// TIA Portal project "PLC_TEST_PROJECT_1" (V16)

(* hardware
DEVICE "S71500/ET200MP station_1"  S7-1500 station
   slot 0: "Rail_0"  Rack  6ES7 590-1***0-0AA0
   slot 1: "PLC_1"  CPU 1518F-4 PN/DP  6ES7 518-4FP00-0AB0  V2.8
      slot 3: "CPU display_1"  6ES7591-1BA00-0AA0
      slot 32768: "PROFINET interface_1"  X1
         slot 32769: "Port_1"  X1 P1
         slot 32770: "Port_2"  X1 P2
      slot 33024: "PROFINET interface_2"  X2
         slot 33025: "Port_1"  X2 P1
      slot 33280: "PROFINET interface GBIT_3"  X3
         slot 33281: "Port_1"  X3 P1
      slot 33536: "DP interface_1"  X4
      slot 34817: "Virtual CP interface port_1"  Virtual CP interface port  Virtual CP interface port
DEVICE "PCSTATION"  SIMATIC PC station
   slot 0: "PC station"  Rail  SIMATIC PC-Station  V1.0
      slot 125: "Stationmanager"  Station_Manager  V6.0.4
   slot 2: "HMI_RT_1"  WinCC RT Professional  6AV2 105-0xxxx-xxxx  16.0.0.0
*)

// ===== PLC "PLC_1"  CPU 1518F-4 PN/DP =====

VAR_GLOBAL   // PLC tag table "Default tag table"
   "Clock_Byte" AT %MB0 : Byte;
   "Clock_10Hz" AT %M0.0 : Bool;
   "Clock_5Hz" AT %M0.1 : Bool;
   "Clock_2.5Hz" AT %M0.2 : Bool;
   "Clock_2Hz" AT %M0.3 : Bool;
   "Clock_1.25Hz" AT %M0.4 : Bool;
   "Clock_1Hz" AT %M0.5 : Bool;
   "Clock_0.625Hz" AT %M0.6 : Bool;
   "Clock_0.5Hz" AT %M0.7 : Bool;
   "Tag_1" AT %MD104 : DWord;
   "Tag_2" AT %MD100 : DWord;
END_VAR

// folder: Common

TYPE "typeDiagnostics"
TITLE = typeDiagnostics
// Provides a structure for detailed diagnostics
   STRUCT
      status : Word;   // Status of the block or error identification when error occurred
      subfunctionStatus : DWord;   // Status or return value of called FBs, FCs and system blocks
      stateNumber : DInt;   // State in the state machine of the block where the error occurred
   END_STRUCT;
END_TYPE

// folder: LMQTT

TYPE "LMQTT_typeConnParam"
TITLE = LMQTT_typeConnParams
// Specifies connection parameters for the mqtt connection
   STRUCT
      hwId : Hw_Any;   // Hardware identifier of the interface. 0: interface is selected automatically
      connId : Conn_Ouc;   // Unique connection identifier
      brokerAddress : Struct   // Information on the MQTT broker
         qdnAddress : String;   // Fully qualified domain name of the broker. must end with a dot "."
         ipAddress : IP_V4;   // If no FQDN is used, enter ip-address of the broker instead
         port : UInt;   // Enter the port of the mqtt broker
      END_STRUCT;
      tls : Struct   // Parameters for TLS encryption
         enableTls : Bool;   // TRUE: Enables TLS, FALSE: disable TLS
         validateServerIdentity : Bool;   // TRUE: Validate server certificate, FALSE: No validation of server certificate
         brokerCert : UDInt;   // ID of the broker's certificate in TIA Portal
         clientCert : UDInt;   // ID of the client's certificate in TIA Portal
      END_STRUCT;
      keepAlive : UInt;   // Keepalive mechanism for MQTT in seconds. 0: disabled.
   END_STRUCT;
END_TYPE

// folder: (top level)

DATA_BLOCK "Main_Safety_RTG1_DB"   // DB1, F_DB
{ S7_Optimized_Access := 'TRUE' }
NAME : FUSI
VERSION : 0.1
// stored: InstanceOfName Main_Safety_RTG1
"Main_Safety_RTG1"
BEGIN
END_DATA_BLOCK

DATA_BLOCK "Timers"   // DB7
{ S7_Optimized_Access := 'TRUE' }
VERSION : 0.1
   VAR
      ElapsedTime : Time;
   END_VAR
BEGIN
END_DATA_BLOCK

DATA_BLOCK "DB_CMD"   // DB100
{ S7_Optimized_Access := 'FALSE' }
VERSION : 0.1
   VAR
      CMD_BOOL_1 : Bool;
      CMD_BOOL_2 : Bool;
      CMD_BOOL_3 : Bool;
      CMD_BOOL_4 : Bool;
      CMD_BOOL_5 : Bool;
      EnableCyclicPub : Bool;
      EnableTimeFrame : Bool;
      CMD_BOOL_8 : Bool;
      CMD_BOOL_9 : Bool;
      CMD_BOOL_10 : Bool;
      EnableCounter : Bool;
      EnableCounter4 : Bool;
      EnableCounter6 : Bool;
      EnableCounter10 : Bool;
   END_VAR
BEGIN
END_DATA_BLOCK

DATA_BLOCK "DB_STATUS"   // DB200
{ S7_Optimized_Access := 'FALSE' }
VERSION : 0.1
   VAR
      STAT_INT_1 : Int;
      STAT_INT_2 : Int;
      STAT_INT_3 : Int;
      STAT_INT_4 : Int;
      STAT_INT_5 : Int;
      STAT_INT_6 : Int;
      STAT_INT_7 : Int;
      STAT_INT_8 : Int;
      STAT_INT_9 : Int;
      STAT_INT_10 : Int;
      STAT_DINT_1 : DInt;
      STAT_DINT_2 : DInt;
      STAT_DINT_3 : DInt;
      STAT_DINT_4 : DInt;
      STAT_DINT_5 : DInt;
      STAT_DINT_6 : DInt;
      STAT_DINT_7 : DInt;
      STAT_DINT_8 : DInt;
      STAT_DINT_9 : DInt;
      STAT_DINT_10 : DInt;
      STAT_BOOL_1 : Bool;
      STAT_BOOL_2 : Bool;
      STAT_BOOL_3 : Bool;
      STAT_BOOL_4 : Bool;
      STAT_BOOL_5 : Bool;
      STAT_BOOL_6 : Bool;
      STAT_BOOL_7 : Bool;
      STAT_BOOL_8 : Bool;
      STAT_BOOL_9 : Bool;
      STAT_BOOL_10 : Bool;
      STAT_WCHAR_1 : Array[0..9] of Char;
   END_VAR
BEGIN
   STAT_WCHAR_1[0] := 'c';
   STAT_WCHAR_1[1] := 'b';
   STAT_WCHAR_1[2] := 'c';
END_DATA_BLOCK

DATA_BLOCK "DB_STATUS_CHECK"   // DB201
{ S7_Optimized_Access := 'FALSE' }
VERSION : 0.1
   VAR
      STAT_INT_1 : Int;
      STAT_INT_2 : Int;
      STAT_INT_3 : Int;
      STAT_INT_4 : Int;
      STAT_INT_5 : Int;
      STAT_INT_6 : Int;
      STAT_INT_7 : Int;
      STAT_INT_8 : Int;
      STAT_INT_9 : Int;
      STAT_INT_10 : Int;
      STAT_DINT_1 : DInt;
      STAT_DINT_2 : DInt;
      STAT_DINT_3 : DInt;
      STAT_DINT_4 : DInt;
      STAT_DINT_5 : DInt;
      STAT_DINT_6 : DInt;
      STAT_DINT_7 : DInt;
      STAT_DINT_8 : DInt;
      STAT_DINT_9 : DInt;
      STAT_DINT_10 : DInt;
      STAT_BOOL_1 : Bool;
      STAT_BOOL_2 : Bool;
      STAT_BOOL_3 : Bool;
      STAT_BOOL_4 : Bool;
      STAT_BOOL_5 : Bool;
      STAT_BOOL_6 : Bool;
      STAT_BOOL_7 : Bool;
      STAT_BOOL_8 : Bool;
      STAT_BOOL_9 : Bool;
      STAT_BOOL_10 : Bool;
      STAT_WCHAR_1 : Array[0..9] of Char;
   END_VAR
BEGIN
   STAT_WCHAR_1[0] := 'c';
   STAT_WCHAR_1[1] := 'b';
   STAT_WCHAR_1[2] := 'c';
END_DATA_BLOCK

DATA_BLOCK "DB_STATUS_ADDR_BYTE"   // DB202
{ S7_Optimized_Access := 'FALSE' }
VERSION : 0.1
   VAR
      STAT_INT_1 : Int := 0;
      STAT_INT_2 : Int := 2;
      STAT_INT_3 : Int := 4;
      STAT_INT_4 : Int := 6;
      STAT_INT_5 : Int := 8;
      STAT_INT_6 : Int := 10;
      STAT_INT_7 : Int := 12;
      STAT_INT_8 : Int := 14;
      STAT_INT_9 : Int := 16;
      STAT_INT_10 : Int := 18;
      STAT_DINT_1 : Int := 20;
      STAT_DINT_2 : Int := 24;
      STAT_DINT_3 : Int := 28;
      STAT_DINT_4 : Int := 32;
      STAT_DINT_5 : Int := 36;
      STAT_DINT_6 : Int := 40;
      STAT_DINT_7 : Int := 44;
      STAT_DINT_8 : Int := 48;
      STAT_DINT_9 : Int := 52;
      STAT_DINT_10 : Int := 56;
      STAT_BOOL_1 : Int := 60;
      STAT_BOOL_2 : Int := 60;
      STAT_BOOL_3 : Int := 60;
      STAT_BOOL_4 : Int := 60;
      STAT_BOOL_5 : Int := 60;
      STAT_BOOL_6 : Int := 60;
      STAT_BOOL_7 : Int := 60;
      STAT_BOOL_8 : Int := 60;
      STAT_BOOL_9 : Int := 61;
      STAT_BOOL_10 : Int := 61;
      STAT_WCHAR_1 : Int := 62;
   END_VAR
BEGIN
END_DATA_BLOCK

DATA_BLOCK "DB_STATUS_ADDR_BIT"   // DB203
{ S7_Optimized_Access := 'FALSE' }
VERSION : 0.1
   VAR
      STAT_INT_1 : Byte := 0;
      STAT_INT_2 : Byte := 0;
      STAT_INT_3 : Byte := 0;
      STAT_INT_4 : Byte := 0;
      STAT_INT_5 : Byte := 0;
      STAT_INT_6 : Byte := 0;
      STAT_INT_7 : Byte := 0;
      STAT_INT_8 : Byte := 0;
      STAT_INT_9 : Byte := 0;
      STAT_INT_10 : Byte := 0;
      STAT_DINT_1 : Byte := 0;
      STAT_DINT_2 : Byte := 0;
      STAT_DINT_3 : Byte := 0;
      STAT_DINT_4 : Byte := 0;
      STAT_DINT_5 : Byte := 0;
      STAT_DINT_6 : Byte := 0;
      STAT_DINT_7 : Byte := 0;
      STAT_DINT_8 : Byte := 0;
      STAT_DINT_9 : Byte := 0;
      STAT_DINT_10 : Byte := 0;
      STAT_BOOL_1 : Byte := 0;
      STAT_BOOL_2 : Byte := 1;
      STAT_BOOL_3 : Byte := 2;
      STAT_BOOL_4 : Byte := 3;
      STAT_BOOL_5 : Byte := 4;
      STAT_BOOL_6 : Byte := 5;
      STAT_BOOL_7 : Byte := 6;
      STAT_BOOL_8 : Byte := 7;
      STAT_BOOL_9 : Byte := 0;
      STAT_BOOL_10 : Byte := 0;
      STAT_WCHAR_1 : Byte := 10;
   END_VAR
BEGIN
END_DATA_BLOCK

// folder: DataChange

DATA_BLOCK "DB_DataChange"   // DB5
{ S7_Optimized_Access := 'FALSE' }
VERSION : 0.1
   VAR
      StartMQTT : Bool;
      DataChanged : Bool;
      DataTypeCode : Array[0..0] of Byte;
   END_VAR
BEGIN
END_DATA_BLOCK

// folder: LMQTT

DATA_BLOCK "LMQTT_Client_DB"   // DB2
{ S7_Optimized_Access := 'TRUE' }
AUTHOR : SUP
FAMILY : LMQTT
VERSION : 3.0
// stored: InstanceOfName LMQTT_Client
"LMQTT_Client"
BEGIN
END_DATA_BLOCK

DATA_BLOCK "MqttDb"   // DB3
TITLE = Configuration Data block example for LMQTT_Client
{ S7_Optimized_Access := 'TRUE' }
AUTHOR : Siemens
FAMILY : LMQTT
VERSION : 1.0
// This block is an example how to control the LMQTT_Client function block
   VAR
      control : Struct   // Input of the FB
         connect : Bool;   // Set TRUE, to establish a connection - set to FALSE to disconnect
         publish : Bool;   // Rising Edge: Sends a message
         subscribe : Bool;   // Rising Edge: Subscribes to a topic
         unsubscribe : Bool;   // Rising Edge: Unsubscribes to a topic
      END_STRUCT;
      output : Struct   // Output Information of the FB
         valid : Bool;   // TRUE: Valid set of output values available at the FB
         done : Bool;   // TRUE: If last Request was successfull
         busy : Bool;   // TRUE: FB is not finished and new output values can be expected
         error : Bool;   // TRUE: An error occurred during the execution of the FB
         status : Word;   // 16#0000 - 16#7FFF: Status of the FB, 16#8000 - 16#FFFF: Error identification
         diagnostics : "typeDiagnostics";   // Diagnostics information of FB (optional)
      END_STRUCT;
      connparams : "LMQTT_typeConnParam";   // Connection Parameters
      clientid : WString[20] := WSTRING#'SiemensClient';   // ClientId with one or more characters
      username : WString[20];   // Username used for connect
      password : WString[20];   // Password used for connect
      willtopic : WString[20] := WSTRING#'willTopic';   // Topic where the last will message is sent
      willMessage : Array[0..99] of Byte;   // Last will message Data - valid bytes in this array must be written in input 'willMsgLen'
      willmesscnt : UInt := 10;   // Valid number of elements in Will Message Data Array. Max 65535 Byte allowed by MQTT Spec.
      qos : USInt := 0;   // Sets QoS 0,1 or 2 for the Publish and Will Message - Subscribe only allows QoS 0 and 1
      topic : WString[100] := WSTRING#'TIA-test-project';   // Mqtt Topic to Publish / Subscribe / Unsubscribe
      message : Array[0..99] of Byte;   // Message Data to Publish - valid bytes in this array must be written in input 'publishMsgLen'
      pubMessageCnt : UDInt := 11;   // Valid number of elements in publish message data Array
      retain : Bool;   // TRUE: Published Message will be set to retain on MQTT broker
      receivedTopic : WString[200] := WSTRING#'TIA-test-project';   // Mqtt Topic of received message
      receivedmessage : Array[0..99] of Byte;   // Mqtt message data that was received - valid bytes in this array indicated by 'receivedMsgDataLen' output
      receivedMsgLen : UDInt;   // Amount of Bytes received in receivedMessage INOUT area
      receivedMsgStatus : USInt;   // 0: No new Message, 1: New valid Message received and available at InOut area, 2: New message, but data is invalid (wrong message len or message could not be copied to InOut received topic or received message)
   END_VAR
BEGIN
   willMessage[0] := 16#6F;
   willMessage[1] := 16#66;
   willMessage[2] := 16#66;
   willMessage[3] := 16#6C;
   willMessage[4] := 16#69;
   willMessage[5] := 16#6E;
   willMessage[6] := 16#65;
   message[1] := 16#65;
   message[2] := 16#6c;
   message[3] := 16#6c;
   message[4] := 16#6f;
   message[5] := 16#20;
   message[6] := 16#77;
   message[7] := 16#6f;
   message[8] := 16#72;
   message[9] := 16#6c;
   message[10] := 16#64;
   message[0] := 16#68;
   connparams.connId := 16#10;
   connparams.brokerAddress.ipAddress.ADDR[1] := 192;
   connparams.brokerAddress.ipAddress.ADDR[2] := 168;
   connparams.brokerAddress.ipAddress.ADDR[3] := 0;
   connparams.brokerAddress.ipAddress.ADDR[4] := 250;
   connparams.brokerAddress.port := 1883;
   connparams.hwId := 64;
   connparams.keepAlive := 100;
END_DATA_BLOCK

// folder: MQTT_pub

DATA_BLOCK "DB_MQTT_PUB"   // DB4
{ S7_Optimized_Access := 'FALSE' }
VERSION : 0.1
   VAR
      DataTypeCodeTemp : Array[0..0] of Byte;
   END_VAR
BEGIN
END_DATA_BLOCK

// folder: Serialize

DATA_BLOCK "DB_Serialize"   // DB1001
{ S7_Optimized_Access := 'TRUE' }
VERSION : 0.1
   VAR
      SERIAL_BYTEARRAY : Array[0..99] of Byte;
      SER_ERROR_CODE : Int;
      SER_START_INDEX : Int;
   END_VAR
BEGIN
END_DATA_BLOCK

// folder: System blocks/Program resources

DATA_BLOCK "TrigDelay"   // DB6
{ S7_Optimized_Access := 'TRUE' }
AUTHOR : Simatic
FAMILY : IEC
NAME : IEC_TMR
VERSION : 1.0
// stored: InstanceOfName IEC_TIMER
"IEC_TIMER"
BEGIN
END_DATA_BLOCK

DATA_BLOCK "IncrementTimer"   // DB8
{ S7_Optimized_Access := 'TRUE' }
AUTHOR : Simatic
FAMILY : IEC
NAME : IEC_TMR
VERSION : 1.0
// stored: InstanceOfName IEC_TIMER
"IEC_TIMER"
BEGIN
END_DATA_BLOCK

// folder: (top level)

FUNCTION_BLOCK "Main_Safety_RTG1"   // FB1, F_FBD
{ S7_Optimized_Access := 'TRUE' }
BEGIN
END_FUNCTION_BLOCK

FUNCTION "DataChange" : Void   // FC3, SCL
{ S7_Optimized_Access := 'TRUE' }
VERSION : 0.1
   VAR_OUTPUT
      DataChanged : Bool;
   END_VAR
   VAR_TEMP
      i : Int;
      TagChanged : Int;
      DataTypeBytelen : Int;
   END_VAR
BEGIN
   (*

   *)

   IF "DB_STATUS".STAT_INT_1 <> "DB_STATUS_CHECK".STAT_INT_1 THEN
       "DB_STATUS_CHECK".STAT_INT_1 := "DB_STATUS".STAT_INT_1;

       //Serialize address byte  - first 4 bytes in MQTT message array [0,1,2,3]
       "Serialize_to_ByteArray"(StartIndexOutputArray := "DB_Serialize".SER_START_INDEX,
                                Input_tag_any_type := "DB_STATUS_ADDR_BYTE".STAT_INT_1,
                                OutputArray => "MqttDb".message,
                                RetVal_error => "DB_Serialize".SER_ERROR_CODE);
       "DB_Serialize".SER_START_INDEX :=  "DB_Serialize".SER_START_INDEX + 4;

       //Serialize address bit (or array length) -  next 1 byte in MQTT message array [4]
       "Serialize_to_ByteArray"(StartIndexOutputArray := "DB_Serialize".SER_START_INDEX,
                                Input_tag_any_type := "DB_STATUS_ADDR_BIT".STAT_INT_1,
                                OutputArray => "MqttDb".message,
                                RetVal_error => "DB_Serialize".SER_ERROR_CODE);
       "DB_Serialize".SER_START_INDEX := "DB_Serialize".SER_START_INDEX + 1;

       //Serialize data type -  next 1 byte in MQTT message array [5]
       "GetDataTypeCode"(DataTypeByteLen=>#DataTypeBytelen,
                         DataTypeCode => "DB_DataChange".DataTypeCode,
                         InOutVariant := "DB_STATUS".STAT_INT_1);
       "MqttDb".message["DB_Serialize".SER_START_INDEX] := "DB_DataChange".DataTypeCode[0];
       "DB_Serialize".SER_START_INDEX := "DB_Serialize".SER_START_INDEX + 1;

       //Serialize tag value -  next 1 byte in MQTT message array [6]
       "Serialize_to_ByteArray"(StartIndexOutputArray := "DB_Serialize".SER_START_INDEX,
                                Input_tag_any_type := "DB_STATUS".STAT_INT_1,
                                OutputArray => "MqttDb".message,
                                RetVal_error => "DB_Serialize".SER_ERROR_CODE);
       //Set index for next tag in MQTT message array
       "DB_Serialize".SER_START_INDEX := "DB_Serialize".SER_START_INDEX + #DataTypeBytelen;
       #TagChanged := #TagChanged + 1;
   END_IF;

   IF "DB_STATUS".STAT_INT_2 <> "DB_STATUS_CHECK".STAT_INT_2 THEN
       "DB_STATUS_CHECK".STAT_INT_2 := "DB_STATUS".STAT_INT_2;

       //Serialize address byte  - first 4 bytes in MQTT message array [0,1,2,3]
       "Serialize_to_ByteArray"(StartIndexOutputArray := "DB_Serialize".SER_START_INDEX,
                                Input_tag_any_type := "DB_STATUS_ADDR_BYTE".STAT_INT_2,
                                OutputArray => "MqttDb".message,
                                RetVal_error => "DB_Serialize".SER_ERROR_CODE);
       "DB_Serialize".SER_START_INDEX := "DB_Serialize".SER_START_INDEX + 4;

       //Serialize address bit (or array length) -  next 1 byte in MQTT message array [4]
       "Serialize_to_ByteArray"(StartIndexOutputArray := "DB_Serialize".SER_START_INDEX,
                                Input_tag_any_type := "DB_STATUS_ADDR_BIT".STAT_INT_2,
                                OutputArray => "MqttDb".message,
                                RetVal_error => "DB_Serialize".SER_ERROR_CODE);
       "DB_Serialize".SER_START_INDEX := "DB_Serialize".SER_START_INDEX + 1;

       //Serialize data type -  next 1 byte in MQTT message array [5]
       "GetDataTypeCode"(DataTypeByteLen => #DataTypeBytelen,
                         DataTypeCode => "DB_DataChange".DataTypeCode,
                         InOutVariant := "DB_STATUS".STAT_INT_2);
       "MqttDb".message["DB_Serialize".SER_START_INDEX] := "DB_DataChange".DataTypeCode[0];
       "DB_Serialize".SER_START_INDEX := "DB_Serialize".SER_START_INDEX + 1;

       //Serialize tag value -  next 1 byte in MQTT message array [6]
       "Serialize_to_ByteArray"(StartIndexOutputArray := "DB_Serialize".SER_START_INDEX,
                                Input_tag_any_type := "DB_STATUS".STAT_INT_2,
                                OutputArray => "MqttDb".message,
                                RetVal_error => "DB_Serialize".SER_ERROR_CODE);
       //Set index for next tag in MQTT message array
       "DB_Serialize".SER_START_INDEX := "DB_Serialize".SER_START_INDEX + #DataTypeBytelen;
       #TagChanged := #TagChanged + 1;
   END_IF;

   IF "DB_STATUS".STAT_INT_3 <> "DB_STATUS_CHECK".STAT_INT_3 THEN
       "DB_STATUS_CHECK".STAT_INT_3 := "DB_STATUS".STAT_INT_3;

       //Serialize address byte  - first 4 bytes in MQTT message array [0,1,2,3]
       "Serialize_to_ByteArray"(StartIndexOutputArray := "DB_Serialize".SER_START_INDEX,
                                Input_tag_any_type := "DB_STATUS_ADDR_BYTE".STAT_INT_3,
                                OutputArray => "MqttDb".message,
                                RetVal_error => "DB_Serialize".SER_ERROR_CODE);
       "DB_Serialize".SER_START_INDEX := "DB_Serialize".SER_START_INDEX + 4;

       //Serialize address bit (or array length) -  next 1 byte in MQTT message array [4]
       "Serialize_to_ByteArray"(StartIndexOutputArray := "DB_Serialize".SER_START_INDEX,
                                Input_tag_any_type := "DB_STATUS_ADDR_BIT".STAT_INT_3,
                                OutputArray => "MqttDb".message,
                                RetVal_error => "DB_Serialize".SER_ERROR_CODE);
       "DB_Serialize".SER_START_INDEX := "DB_Serialize".SER_START_INDEX + 1;

       //Serialize data type -  next 1 byte in MQTT message array [5]
       "GetDataTypeCode"(DataTypeByteLen => #DataTypeBytelen,
                         DataTypeCode => "DB_DataChange".DataTypeCode,
                         InOutVariant := "DB_STATUS".STAT_INT_3);
       "MqttDb".message["DB_Serialize".SER_START_INDEX] := "DB_DataChange".DataTypeCode[0];
       "DB_Serialize".SER_START_INDEX := "DB_Serialize".SER_START_INDEX + 1;

       //Serialize tag value -  next 1 byte in MQTT message array [6]
       "Serialize_to_ByteArray"(StartIndexOutputArray := "DB_Serialize".SER_START_INDEX,
                                Input_tag_any_type := "DB_STATUS".STAT_INT_3,
                                OutputArray => "MqttDb".message,
                                RetVal_error => "DB_Serialize".SER_ERROR_CODE);
       //Set index for next tag in MQTT message array
       "DB_Serialize".SER_START_INDEX := "DB_Serialize".SER_START_INDEX + #DataTypeBytelen;
       #TagChanged := #TagChanged + 1;
   END_IF;

   IF "DB_STATUS".STAT_INT_4 <> "DB_STATUS_CHECK".STAT_INT_4 THEN
       "DB_STATUS_CHECK".STAT_INT_4 := "DB_STATUS".STAT_INT_4;

       //Serialize address byte  - first 4 bytes in MQTT message array [0,1,2,3]
       "Serialize_to_ByteArray"(StartIndexOutputArray := "DB_Serialize".SER_START_INDEX,
                                Input_tag_any_type := "DB_STATUS_ADDR_BYTE".STAT_INT_4,
                                OutputArray => "MqttDb".message,
                                RetVal_error => "DB_Serialize".SER_ERROR_CODE);
       "DB_Serialize".SER_START_INDEX := "DB_Serialize".SER_START_INDEX + 4;

       //Serialize address bit (or array length) -  next 1 byte in MQTT message array [4]
       "Serialize_to_ByteArray"(StartIndexOutputArray := "DB_Serialize".SER_START_INDEX,
                                Input_tag_any_type := "DB_STATUS_ADDR_BIT".STAT_INT_4,
                                OutputArray => "MqttDb".message,
                                RetVal_error => "DB_Serialize".SER_ERROR_CODE);
       "DB_Serialize".SER_START_INDEX := "DB_Serialize".SER_START_INDEX + 1;

       //Serialize data type -  next 1 byte in MQTT message array [5]
       "GetDataTypeCode"(DataTypeByteLen => #DataTypeBytelen,
                         DataTypeCode => "DB_DataChange".DataTypeCode,
                         InOutVariant := "DB_STATUS".STAT_INT_4);
       "MqttDb".message["DB_Serialize".SER_START_INDEX] := "DB_DataChange".DataTypeCode[0];
       "DB_Serialize".SER_START_INDEX := "DB_Serialize".SER_START_INDEX + 1;

       //Serialize tag value -  next 1 byte in MQTT message array [6]
       "Serialize_to_ByteArray"(StartIndexOutputArray := "DB_Serialize".SER_START_INDEX,
                                Input_tag_any_type := "DB_STATUS".STAT_INT_4,
                                OutputArray => "MqttDb".message,
                                RetVal_error => "DB_Serialize".SER_ERROR_CODE);
       //Set index for next tag in MQTT message array
       "DB_Serialize".SER_START_INDEX := "DB_Serialize".SER_START_INDEX + #DataTypeBytelen;
       #TagChanged := #TagChanged + 1;
   END_IF;

   IF "DB_STATUS".STAT_INT_5 <> "DB_STATUS_CHECK".STAT_INT_5 THEN
       "DB_STATUS_CHECK".STAT_INT_5 := "DB_STATUS".STAT_INT_5;

       //Serialize address byte  - first 4 bytes in MQTT message array [0,1,2,3]
       "Serialize_to_ByteArray"(StartIndexOutputArray := "DB_Serialize".SER_START_INDEX,
                                Input_tag_any_type := "DB_STATUS_ADDR_BYTE".STAT_INT_5,
                                OutputArray => "MqttDb".message,
                                RetVal_error => "DB_Serialize".SER_ERROR_CODE);
       "DB_Serialize".SER_START_INDEX := "DB_Serialize".SER_START_INDEX + 4;

       //Serialize address bit (or array length) -  next 1 byte in MQTT message array [4]
       "Serialize_to_ByteArray"(StartIndexOutputArray := "DB_Serialize".SER_START_INDEX,
                                Input_tag_any_type := "DB_STATUS_ADDR_BIT".STAT_INT_5,
                                OutputArray => "MqttDb".message,
                                RetVal_error => "DB_Serialize".SER_ERROR_CODE);
       "DB_Serialize".SER_START_INDEX := "DB_Serialize".SER_START_INDEX + 1;

       //Serialize data type -  next 1 byte in MQTT message array [5]
       "GetDataTypeCode"(DataTypeByteLen => #DataTypeBytelen,
                         DataTypeCode => "DB_DataChange".DataTypeCode,
                         InOutVariant := "DB_STATUS".STAT_INT_5);
       "MqttDb".message["DB_Serialize".SER_START_INDEX] := "DB_DataChange".DataTypeCode[0];
       "DB_Serialize".SER_START_INDEX := "DB_Serialize".SER_START_INDEX + 1;

       //Serialize tag value -  next 1 byte in MQTT message array [6]
       "Serialize_to_ByteArray"(StartIndexOutputArray := "DB_Serialize".SER_START_INDEX,
                                Input_tag_any_type := "DB_STATUS".STAT_INT_5,
                                OutputArray => "MqttDb".message,
                                RetVal_error => "DB_Serialize".SER_ERROR_CODE);
       //Set index for next tag in MQTT message array
       "DB_Serialize".SER_START_INDEX := "DB_Serialize".SER_START_INDEX + #DataTypeBytelen;
       #TagChanged := #TagChanged + 1;
   END_IF;

   IF "DB_STATUS".STAT_DINT_1 <> "DB_STATUS_CHECK".STAT_DINT_1 THEN
       "DB_STATUS_CHECK".STAT_DINT_1 := "DB_STATUS".STAT_DINT_1;

       //Serialize address byte  - first 4 bytes in MQTT message array [0,1,2,3]
       "Serialize_to_ByteArray"(StartIndexOutputArray := "DB_Serialize".SER_START_INDEX,
                                Input_tag_any_type := "DB_STATUS_ADDR_BYTE".STAT_DINT_1,
                                OutputArray => "MqttDb".message,
                                RetVal_error => "DB_Serialize".SER_ERROR_CODE);
       "DB_Serialize".SER_START_INDEX := "DB_Serialize".SER_START_INDEX + 4;

       //Serialize address bit (or array length) -  next 1 byte in MQTT message array [4]
       "Serialize_to_ByteArray"(StartIndexOutputArray := "DB_Serialize".SER_START_INDEX,
                                Input_tag_any_type := "DB_STATUS_ADDR_BIT".STAT_DINT_1,
                                OutputArray => "MqttDb".message,
                                RetVal_error => "DB_Serialize".SER_ERROR_CODE);
       "DB_Serialize".SER_START_INDEX := "DB_Serialize".SER_START_INDEX + 1;

       //Serialize data type -  next 1 byte in MQTT message array [5]
       "GetDataTypeCode"(DataTypeByteLen => #DataTypeBytelen,
                         DataTypeCode => "DB_DataChange".DataTypeCode,
                         InOutVariant := "DB_STATUS".STAT_DINT_1);
       "MqttDb".message["DB_Serialize".SER_START_INDEX] := "DB_DataChange".DataTypeCode[0];
       "DB_Serialize".SER_START_INDEX := "DB_Serialize".SER_START_INDEX + 1;

       //Serialize tag value -  next 1 byte in MQTT message array [6]
       "Serialize_to_ByteArray"(StartIndexOutputArray := "DB_Serialize".SER_START_INDEX,
                                Input_tag_any_type := "DB_STATUS".STAT_DINT_1,
                                OutputArray => "MqttDb".message,
                                RetVal_error => "DB_Serialize".SER_ERROR_CODE);
       //Set index for next tag in MQTT message array
       "DB_Serialize".SER_START_INDEX := "DB_Serialize".SER_START_INDEX + #DataTypeBytelen;
       #TagChanged := #TagChanged + 1;
   END_IF;

   IF "DB_STATUS".STAT_DINT_2 <> "DB_STATUS_CHECK".STAT_DINT_2 THEN
       "DB_STATUS_CHECK".STAT_DINT_2 := "DB_STATUS".STAT_DINT_2;

       //Serialize address byte  - first 4 bytes in MQTT message array [0,1,2,3]
       "Serialize_to_ByteArray"(StartIndexOutputArray := "DB_Serialize".SER_START_INDEX,
                                Input_tag_any_type := "DB_STATUS_ADDR_BYTE".STAT_DINT_2,
                                OutputArray => "MqttDb".message,
                                RetVal_error => "DB_Serialize".SER_ERROR_CODE);
       "DB_Serialize".SER_START_INDEX := "DB_Serialize".SER_START_INDEX + 4;

       //Serialize address bit (or array length) -  next 1 byte in MQTT message array [4]
       "Serialize_to_ByteArray"(StartIndexOutputArray := "DB_Serialize".SER_START_INDEX,
                                Input_tag_any_type := "DB_STATUS_ADDR_BIT".STAT_DINT_2,
                                OutputArray => "MqttDb".message,
                                RetVal_error => "DB_Serialize".SER_ERROR_CODE);
       "DB_Serialize".SER_START_INDEX := "DB_Serialize".SER_START_INDEX + 1;

       //Serialize data type -  next 1 byte in MQTT message array [5]
       "GetDataTypeCode"(DataTypeByteLen => #DataTypeBytelen,
                         DataTypeCode => "DB_DataChange".DataTypeCode,
                         InOutVariant := "DB_STATUS".STAT_DINT_2);
       "MqttDb".message["DB_Serialize".SER_START_INDEX] := "DB_DataChange".DataTypeCode[0];
       "DB_Serialize".SER_START_INDEX := "DB_Serialize".SER_START_INDEX + 1;

       //Serialize tag value -  next 1 byte in MQTT message array [6]
       "Serialize_to_ByteArray"(StartIndexOutputArray := "DB_Serialize".SER_START_INDEX,
                                Input_tag_any_type := "DB_STATUS".STAT_DINT_2,
                                OutputArray => "MqttDb".message,
                                RetVal_error => "DB_Serialize".SER_ERROR_CODE);
       //Set index for next tag in MQTT message array
       "DB_Serialize".SER_START_INDEX := "DB_Serialize".SER_START_INDEX + #DataTypeBytelen;
       #TagChanged := #TagChanged + 1;
   END_IF;

   IF "DB_STATUS".STAT_DINT_3 <> "DB_STATUS_CHECK".STAT_DINT_3 THEN
       "DB_STATUS_CHECK".STAT_DINT_3 := "DB_STATUS".STAT_DINT_3;

       //Serialize address byte  - first 4 bytes in MQTT message array [0,1,2,3]
       "Serialize_to_ByteArray"(StartIndexOutputArray := "DB_Serialize".SER_START_INDEX,
                                Input_tag_any_type := "DB_STATUS_ADDR_BYTE".STAT_DINT_3,
                                OutputArray => "MqttDb".message,
                                RetVal_error => "DB_Serialize".SER_ERROR_CODE);
       "DB_Serialize".SER_START_INDEX := "DB_Serialize".SER_START_INDEX + 4;

       //Serialize address bit (or array length) -  next 1 byte in MQTT message array [4]
       "Serialize_to_ByteArray"(StartIndexOutputArray := "DB_Serialize".SER_START_INDEX,
                                Input_tag_any_type := "DB_STATUS_ADDR_BIT".STAT_DINT_3,
                                OutputArray => "MqttDb".message,
                                RetVal_error => "DB_Serialize".SER_ERROR_CODE);
       "DB_Serialize".SER_START_INDEX := "DB_Serialize".SER_START_INDEX + 1;

       //Serialize data type -  next 1 byte in MQTT message array [5]
       "GetDataTypeCode"(DataTypeByteLen => #DataTypeBytelen,
                         DataTypeCode => "DB_DataChange".DataTypeCode,
                         InOutVariant := "DB_STATUS".STAT_DINT_3);
       "MqttDb".message["DB_Serialize".SER_START_INDEX] := "DB_DataChange".DataTypeCode[0];
       "DB_Serialize".SER_START_INDEX := "DB_Serialize".SER_START_INDEX + 1;

       //Serialize tag value -  next 1 byte in MQTT message array [6]
       "Serialize_to_ByteArray"(StartIndexOutputArray := "DB_Serialize".SER_START_INDEX,
                                Input_tag_any_type := "DB_STATUS".STAT_DINT_3,
                                OutputArray => "MqttDb".message,
                                RetVal_error => "DB_Serialize".SER_ERROR_CODE);
       //Set index for next tag in MQTT message array
       "DB_Serialize".SER_START_INDEX := "DB_Serialize".SER_START_INDEX + #DataTypeBytelen;
       #TagChanged := #TagChanged + 1;
   END_IF;

   IF "DB_STATUS".STAT_DINT_4 <> "DB_STATUS_CHECK".STAT_DINT_4 THEN
       "DB_STATUS_CHECK".STAT_DINT_4 := "DB_STATUS".STAT_DINT_4;

       //Serialize address byte  - first 4 bytes in MQTT message array [0,1,2,3]
       "Serialize_to_ByteArray"(StartIndexOutputArray := "DB_Serialize".SER_START_INDEX,
                                Input_tag_any_type := "DB_STATUS_ADDR_BYTE".STAT_DINT_4,
                                OutputArray => "MqttDb".message,
                                RetVal_error => "DB_Serialize".SER_ERROR_CODE);
       "DB_Serialize".SER_START_INDEX := "DB_Serialize".SER_START_INDEX + 4;

       //Serialize address bit (or array length) -  next 1 byte in MQTT message array [4]
       "Serialize_to_ByteArray"(StartIndexOutputArray := "DB_Serialize".SER_START_INDEX,
                                Input_tag_any_type := "DB_STATUS_ADDR_BIT".STAT_DINT_4,
                                OutputArray => "MqttDb".message,
                                RetVal_error => "DB_Serialize".SER_ERROR_CODE);
       "DB_Serialize".SER_START_INDEX := "DB_Serialize".SER_START_INDEX + 1;

       //Serialize data type -  next 1 byte in MQTT message array [5]
       "GetDataTypeCode"(DataTypeByteLen => #DataTypeBytelen,
                         DataTypeCode => "DB_DataChange".DataTypeCode,
                         InOutVariant := "DB_STATUS".STAT_DINT_4);
       "MqttDb".message["DB_Serialize".SER_START_INDEX] := "DB_DataChange".DataTypeCode[0];
       "DB_Serialize".SER_START_INDEX := "DB_Serialize".SER_START_INDEX + 1;

       //Serialize tag value -  next 1 byte in MQTT message array [6]
       "Serialize_to_ByteArray"(StartIndexOutputArray := "DB_Serialize".SER_START_INDEX,
                                Input_tag_any_type := "DB_STATUS".STAT_DINT_4,
                                OutputArray => "MqttDb".message,
                                RetVal_error => "DB_Serialize".SER_ERROR_CODE);
       //Set index for next tag in MQTT message array
       "DB_Serialize".SER_START_INDEX := "DB_Serialize".SER_START_INDEX + #DataTypeBytelen;
       #TagChanged := #TagChanged + 1;
   END_IF;

   IF "DB_STATUS".STAT_DINT_5 <> "DB_STATUS_CHECK".STAT_DINT_5 THEN
       "DB_STATUS_CHECK".STAT_DINT_5 := "DB_STATUS".STAT_DINT_5;

       //Serialize address byte  - first 4 bytes in MQTT message array [0,1,2,3]
       "Serialize_to_ByteArray"(StartIndexOutputArray := "DB_Serialize".SER_START_INDEX,
                                Input_tag_any_type := "DB_STATUS_ADDR_BYTE".STAT_DINT_5,
                                OutputArray => "MqttDb".message,
                                RetVal_error => "DB_Serialize".SER_ERROR_CODE);
       "DB_Serialize".SER_START_INDEX := "DB_Serialize".SER_START_INDEX + 4;

       //Serialize address bit (or array length) -  next 1 byte in MQTT message array [4]
       "Serialize_to_ByteArray"(StartIndexOutputArray := "DB_Serialize".SER_START_INDEX,
                                Input_tag_any_type := "DB_STATUS_ADDR_BIT".STAT_DINT_5,
                                OutputArray => "MqttDb".message,
                                RetVal_error => "DB_Serialize".SER_ERROR_CODE);
       "DB_Serialize".SER_START_INDEX := "DB_Serialize".SER_START_INDEX + 1;

       //Serialize data type -  next 1 byte in MQTT message array [5]
       "GetDataTypeCode"(DataTypeByteLen => #DataTypeBytelen,
                         DataTypeCode => "DB_DataChange".DataTypeCode,
                         InOutVariant := "DB_STATUS".STAT_DINT_5);
       "MqttDb".message["DB_Serialize".SER_START_INDEX] := "DB_DataChange".DataTypeCode[0];
       "DB_Serialize".SER_START_INDEX := "DB_Serialize".SER_START_INDEX + 1;

       //Serialize tag value -  next 1 byte in MQTT message array [6]
       "Serialize_to_ByteArray"(StartIndexOutputArray := "DB_Serialize".SER_START_INDEX,
                                Input_tag_any_type := "DB_STATUS".STAT_DINT_5,
                                OutputArray => "MqttDb".message,
                                RetVal_error => "DB_Serialize".SER_ERROR_CODE);
       //Set index for next tag in MQTT message array
       "DB_Serialize".SER_START_INDEX := "DB_Serialize".SER_START_INDEX + #DataTypeBytelen;
       #TagChanged := #TagChanged + 1;
   END_IF;

   IF "DB_STATUS".STAT_DINT_6 <> "DB_STATUS_CHECK".STAT_DINT_6 THEN
       "DB_STATUS_CHECK".STAT_DINT_6 := "DB_STATUS".STAT_DINT_6;

       //Serialize address byte  - first 4 bytes in MQTT message array [0,1,2,3]
       "Serialize_to_ByteArray"(StartIndexOutputArray := "DB_Serialize".SER_START_INDEX,
                                Input_tag_any_type := "DB_STATUS_ADDR_BYTE".STAT_DINT_6,
                                OutputArray => "MqttDb".message,
                                RetVal_error => "DB_Serialize".SER_ERROR_CODE);
       "DB_Serialize".SER_START_INDEX := "DB_Serialize".SER_START_INDEX + 4;

       //Serialize address bit (or array length) -  next 1 byte in MQTT message array [4]
       "Serialize_to_ByteArray"(StartIndexOutputArray := "DB_Serialize".SER_START_INDEX,
                                Input_tag_any_type := "DB_STATUS_ADDR_BIT".STAT_DINT_6,
                                OutputArray => "MqttDb".message,
                                RetVal_error => "DB_Serialize".SER_ERROR_CODE);
       "DB_Serialize".SER_START_INDEX := "DB_Serialize".SER_START_INDEX + 1;

       //Serialize data type -  next 1 byte in MQTT message array [5]
       "GetDataTypeCode"(DataTypeByteLen => #DataTypeBytelen,
                         DataTypeCode => "DB_DataChange".DataTypeCode,
                         InOutVariant := "DB_STATUS".STAT_DINT_6);
       "MqttDb".message["DB_Serialize".SER_START_INDEX] := "DB_DataChange".DataTypeCode[0];
       "DB_Serialize".SER_START_INDEX := "DB_Serialize".SER_START_INDEX + 1;

       //Serialize tag value -  next 1 byte in MQTT message array [6]
       "Serialize_to_ByteArray"(StartIndexOutputArray := "DB_Serialize".SER_START_INDEX,
                                Input_tag_any_type := "DB_STATUS".STAT_DINT_6,
                                OutputArray => "MqttDb".message,
                                RetVal_error => "DB_Serialize".SER_ERROR_CODE);
       //Set index for next tag in MQTT message array
       "DB_Serialize".SER_START_INDEX := "DB_Serialize".SER_START_INDEX + #DataTypeBytelen;
       #TagChanged := #TagChanged + 1;
   END_IF;

   //If any of the tags are changed, set output trigger.
   IF #TagChanged > 0 THEN
       "MqttDb".pubMessageCnt := "DB_Serialize".SER_START_INDEX; //Message array size
       "MqttDb".topic := WSTRING#'TIA-test-project/DB200';
       #DataChanged := TRUE;
   END_IF;
END_FUNCTION

ORGANIZATION_BLOCK "Main"   // OB1, LAD, ProgramCycle
TITLE = "Main Program Sweep (Cycle)"
{ S7_Optimized_Access := 'TRUE' }
VERSION : 0.1
   VAR_INPUT
      Initial_Call : Bool;   // Initial call of this OB
      Remanence : Bool;   // =True, if remanent data are available
   END_VAR
   VAR_TEMP   // added for the SCL form of the ladder/FBD networks
      _w1 : Bool;
      _w2 : Bool;
   END_VAR
BEGIN

REGION Network 1
   // MQTT client
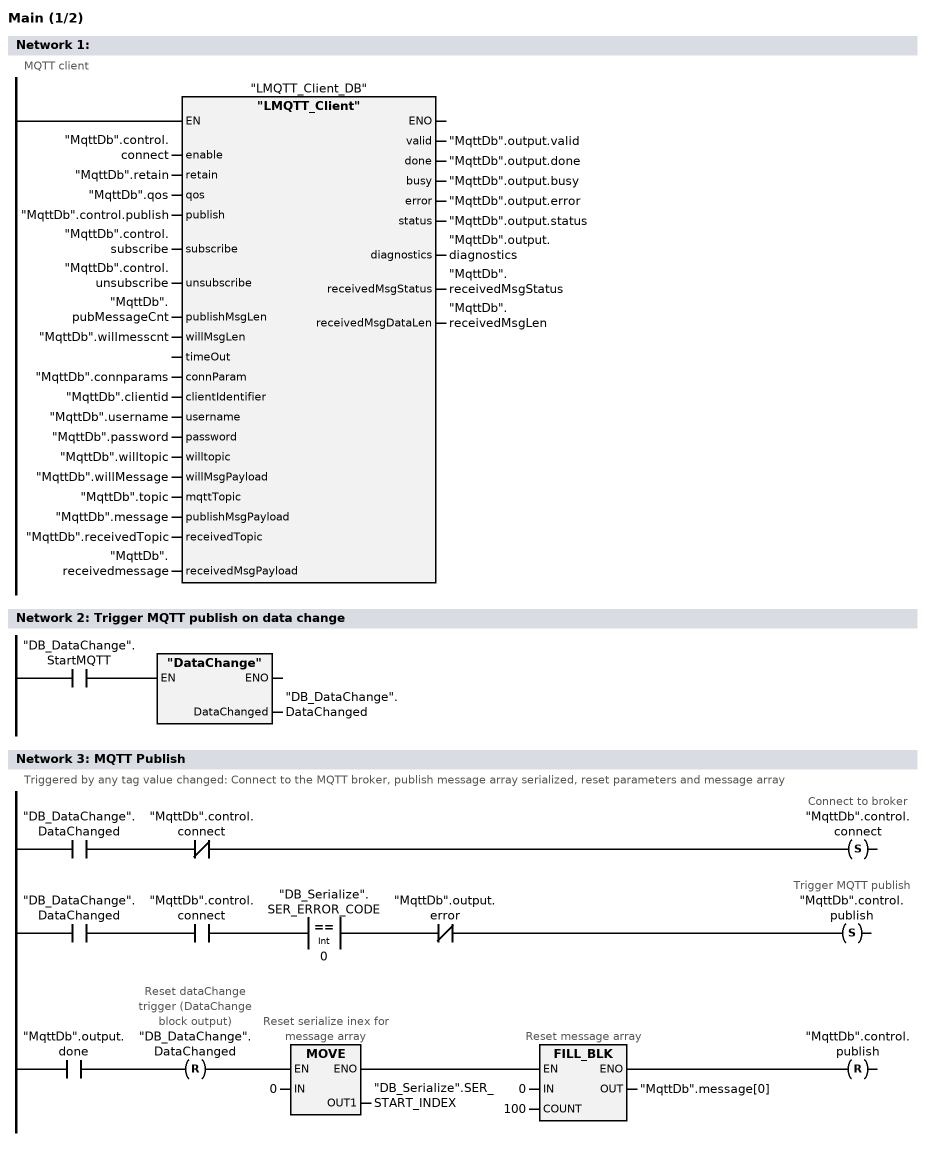
   RUNG wire#powerrail
      "LMQTT_Client_DB"(enable := "MqttDb".control.connect, retain := "MqttDb".retain, qos := "MqttDb".qos, publish := "MqttDb".control.publish, subscribe := "MqttDb".control.subscribe, unsubscribe := "MqttDb".control.unsubscribe, publishMsgLen := "MqttDb".pubMessageCnt, willMsgLen := "MqttDb".willmesscnt, timeOut :=, connParam := "MqttDb".connparams, clientIdentifier := "MqttDb".clientid, username := "MqttDb".username, password := "MqttDb".password, willtopic := "MqttDb".willtopic, willMsgPayload := "MqttDb".willMessage, mqttTopic := "MqttDb".topic, publishMsgPayload := "MqttDb".message, receivedTopic := "MqttDb".receivedTopic, receivedMsgPayload := "MqttDb".receivedmessage, valid => "MqttDb".output.valid, done => "MqttDb".output.done, busy => "MqttDb".output.busy, error => "MqttDb".output.error, status => "MqttDb".output.status, diagnostics => "MqttDb".output.diagnostics, receivedMsgStatus => "MqttDb".receivedMsgStatus, receivedMsgDataLen => "MqttDb".receivedMsgLen)
   END_RUNG
   // the same network as SCL:
   "LMQTT_Client_DB"(enable := "MqttDb".control.connect,   // "LMQTT_Client"
                     retain := "MqttDb".retain,
                     qos := "MqttDb".qos,
                     publish := "MqttDb".control.publish,
                     subscribe := "MqttDb".control.subscribe,
                     unsubscribe := "MqttDb".control.unsubscribe,
                     publishMsgLen := "MqttDb".pubMessageCnt,
                     willMsgLen := "MqttDb".willmesscnt,
                     connParam := "MqttDb".connparams,
                     clientIdentifier := "MqttDb".clientid,
                     username := "MqttDb".username,
                     password := "MqttDb".password,
                     willtopic := "MqttDb".willtopic,
                     willMsgPayload := "MqttDb".willMessage,
                     mqttTopic := "MqttDb".topic,
                     publishMsgPayload := "MqttDb".message,
                     receivedTopic := "MqttDb".receivedTopic,
                     receivedMsgPayload := "MqttDb".receivedmessage,
                     valid => "MqttDb".output.valid,
                     done => "MqttDb".output.done,
                     busy => "MqttDb".output.busy,
                     error => "MqttDb".output.error,
                     status => "MqttDb".output.status,
                     diagnostics => "MqttDb".output.diagnostics,
                     receivedMsgStatus => "MqttDb".receivedMsgStatus,
                     receivedMsgDataLen => "MqttDb".receivedMsgLen);
END_REGION

REGION Network 2: Trigger MQTT publish on data change
   RUNG wire#powerrail
      Contact( "DB_DataChange".StartMQTT )
      "DataChange"(DataChanged => "DB_DataChange".DataChanged)
   END_RUNG
   // the same network as SCL:
   IF "DB_DataChange".StartMQTT THEN "DataChange"(DataChanged => "DB_DataChange".DataChanged); END_IF;
END_REGION

REGION Network 3: MQTT Publish
   // Triggered by any tag value changed: Connect to the MQTT broker, publish message array serialized, reset parameters and message array
   RUNG wire#powerrail
      Contact( "DB_DataChange".DataChanged )
      I_Contact( "MqttDb".control.connect )
      S_Coil( "MqttDb".control.connect )   // Connect to broker
   END_RUNG
   RUNG wire#powerrail
      Contact( "DB_DataChange".DataChanged )
      Contact( "MqttDb".control.connect )
      { S7_Templates := "SrcType := Int" } EQ_Contact(in1 := "DB_Serialize".SER_ERROR_CODE, in2 := 0)
      I_Contact( "MqttDb".output.error )
      S_Coil( "MqttDb".control.publish )   // Trigger MQTT publish
   END_RUNG
   RUNG wire#powerrail
      Contact( "MqttDb".output.done )
      R_Coil( "DB_DataChange".DataChanged )   // Reset dataChange trigger (DataChange block output)
      Move(in := 0, out1 => "DB_Serialize".SER_START_INDEX)   // Reset serialize inex for message array
      FillBlockI(in := 0, count := 100, out => "MqttDb".message[0])   // Reset message array
      R_Coil( "MqttDb".control.publish )
   END_RUNG
   // the same network as SCL:
   IF "DB_DataChange".DataChanged AND NOT "MqttDb".control.connect THEN
       "MqttDb".control.connect := TRUE;   // Connect to broker
   END_IF;
   IF "DB_DataChange".DataChanged AND "MqttDb".control.connect AND ("DB_Serialize".SER_ERROR_CODE = 0) AND NOT "MqttDb".output.error THEN
       "MqttDb".control.publish := TRUE;   // Trigger MQTT publish
   END_IF;
   IF "MqttDb".output.done THEN
       "DB_DataChange".DataChanged := FALSE;   // Reset dataChange trigger (DataChange block output)
       "DB_Serialize".SER_START_INDEX := 0;   // Reset serialize inex for message array
   END_IF;
   #_w1 := "MqttDb".output.done;
   IF #_w1 THEN
       FILL_BLK(IN := 0, COUNT := 100, OUT => "MqttDb".message[0]);   // Reset message array
       "MqttDb".control.publish := FALSE;
   END_IF;
END_REGION

REGION Network 4: Testing area
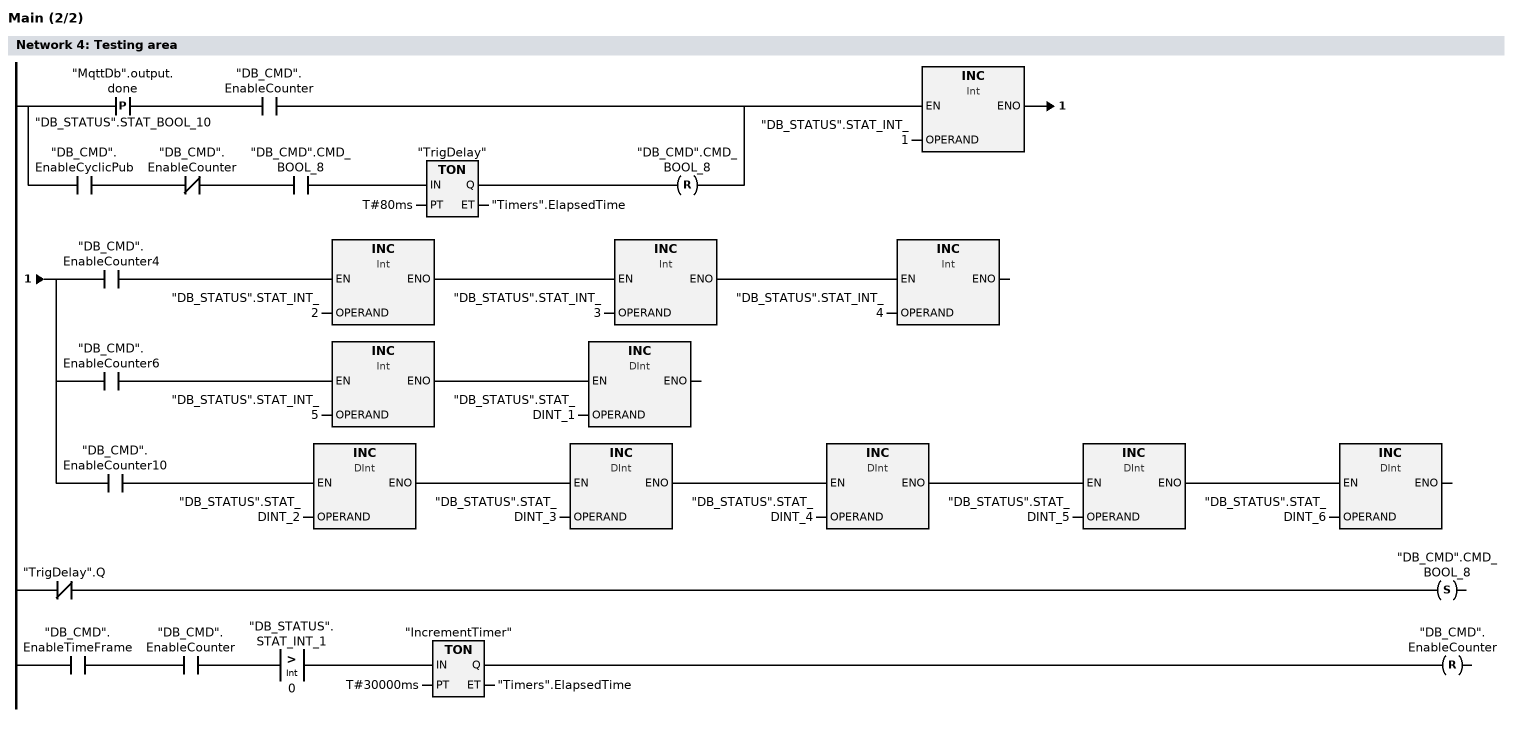
   #_w1 := "MqttDb".output.done AND NOT "DB_STATUS".STAT_BOOL_10;   // rising edge of "MqttDb".output.done
   "DB_STATUS".STAT_BOOL_10 := "MqttDb".output.done;
   "TrigDelay".TON(IN := "DB_CMD".EnableCyclicPub AND NOT "DB_CMD".EnableCounter AND "DB_CMD".CMD_BOOL_8,
                   PT := T#80ms,
                   ET => "Timers".ElapsedTime);
   IF "TrigDelay".Q THEN "DB_CMD".CMD_BOOL_8 := FALSE; END_IF;
   #_w2 := (#_w1 AND "DB_CMD".EnableCounter) OR "TrigDelay".Q;
   IF #_w2 THEN "DB_STATUS".STAT_INT_1 := "DB_STATUS".STAT_INT_1 + 1; END_IF;
   IF #_w2 AND "DB_CMD".EnableCounter4 THEN
       "DB_STATUS".STAT_INT_2 := "DB_STATUS".STAT_INT_2 + 1;
       "DB_STATUS".STAT_INT_3 := "DB_STATUS".STAT_INT_3 + 1;
       "DB_STATUS".STAT_INT_4 := "DB_STATUS".STAT_INT_4 + 1;
   END_IF;
   IF #_w2 AND "DB_CMD".EnableCounter6 THEN
       "DB_STATUS".STAT_INT_5 := "DB_STATUS".STAT_INT_5 + 1;
       "DB_STATUS".STAT_DINT_1 := "DB_STATUS".STAT_DINT_1 + 1;
   END_IF;
   IF #_w2 AND "DB_CMD".EnableCounter10 THEN
       "DB_STATUS".STAT_DINT_2 := "DB_STATUS".STAT_DINT_2 + 1;
       "DB_STATUS".STAT_DINT_3 := "DB_STATUS".STAT_DINT_3 + 1;
       "DB_STATUS".STAT_DINT_4 := "DB_STATUS".STAT_DINT_4 + 1;
       "DB_STATUS".STAT_DINT_5 := "DB_STATUS".STAT_DINT_5 + 1;
       "DB_STATUS".STAT_DINT_6 := "DB_STATUS".STAT_DINT_6 + 1;
   END_IF;
   IF NOT "TrigDelay".Q THEN "DB_CMD".CMD_BOOL_8 := TRUE; END_IF;
   "IncrementTimer".TON(IN := "DB_CMD".EnableTimeFrame AND "DB_CMD".EnableCounter AND ("DB_STATUS".STAT_INT_1 > 0),
                        PT := T#30000ms,
                        ET => "Timers".ElapsedTime);
   IF "IncrementTimer".Q THEN "DB_CMD".EnableCounter := FALSE; END_IF;
END_REGION
END_ORGANIZATION_BLOCK

// folder: LMQTT

FUNCTION_BLOCK "LMQTT_Client"   // FB11, SCL
TITLE = LMQTT_Client
{ S7_Optimized_Access := 'TRUE' }
AUTHOR : SUP
FAMILY : LMQTT
VERSION : 3.0
// This block allows to connect to an MQTT Broker and publish data or receive data via a subscription.
   VAR_INPUT
      enable : Bool;   // Set TRUE, to establish a connection - set to FALSE to disconnect
      retain : Bool;   // TRUE: Published Message will be set to retain on MQTT broker
      qos : USInt;   // Quality of Service for publish/subscribe requests and last will. Subscribe only allows QoS 0 and 1 / Sets QoS 0,1 or 2 for the Publish and Will Message - Subscribe only allows QoS 0 and 1
      publish : Bool;   // Rising Edge: Sends a message
      subscribe : Bool;   // Rising Edge: Subscribes to a topic
      unsubscribe : Bool;   // Rising Edge: Unsubscribes to a topic
      publishMsgLen : UDInt;   // Valid number of elements in publish message data Array
      willMsgLen : UInt;   // Valid number of elements in Will Message Data Array. Max 65535 Byte allowed by MQTT Spec.
      timeOut : Time := T#15s;   // Sets the time out value for every request (publish/subscribe/unsubscribe/ping)
   END_VAR
   VAR_OUTPUT
      valid : Bool;   // TRUE: Valid set of output values available at the FB
      done : Bool;   // TRUE: If last Request was successfull
      busy : Bool;   // TRUE: FB is not finished and new output values can be expected
      error : Bool;   // TRUE: An error occurred during the execution of the FB
      status : Word := 16#7000;   // 16#0000 - 16#7FFF: Status of the FB, 16#8000 - 16#FFFF: Error identification
      diagnostics : "typeDiagnostics";   // Diagnostics information of FB
      receivedMsgStatus : USInt;   // 0: No new Message, 1: New valid Message received and available at InOut area, 2: New message, but data is invalid (wrong message len or message could not be copied to InOut received topic or received message)
      receivedMsgDataLen : UDInt;   // Amount of Bytes received in receivedMessage INOUT area
   END_VAR
   VAR_IN_OUT
      connParam : "LMQTT_typeConnParam";   // Connection Parameters
      clientIdentifier : WString;   // ClientId with one or more characters
      username : WString;   // Username to connect
      password : WString;   // Password to connect
      willtopic : WString;   // Topic where the last will message is sent
      willMsgPayload : Array[*] of Byte;   // Last will message Data - valid bytes in this array must be written in input 'willMsgLen'
      mqttTopic : WString;   // Mqtt Topic to Publish / Subscribe / Unsubscribe
      publishMsgPayload : Array[*] of Byte;   // Message Data to Publish - valid bytes in this array must be written in input 'publishMsgLen'
      receivedTopic : WString;   // Mqtt Topic of received message
      receivedMsgPayload : Array[*] of Byte;   // Mqtt message data that was received - valid bytes in this array indicated by 'receivedMsgDataLen' output
   END_VAR
   VAR
      statEnableOld : Bool;   // Old value of 'enable' input for edge detection
      statValid : Bool;   // Static value for output 'valid'
      statBusy : Bool;   // Static value for output 'busy'
      statError : Bool;   // Static value for output 'error'
      statErrorUserCleared : Bool;   // Error occurred that can only be solved by user; rising edge at enable input necessary
      statErrorAutoCleared : Bool;   // Error occurred that can be acknowledged by FB
      statStatus : Word := 16#7000;   // Static value for output 'status'
      statDone : Bool;   // Static value for output 'done'
      statRcvMsgStatus : USInt;   // Static value for output 'receivedMsgStatus'
      statRcvMsgDataLen : UDInt;   // Static value for output 'receivedMsgDataLen'
      statSubfunctionStatus : Word;   // Status or return value of called FBs, FCs and system blocks
      statFBErrorState : DInt;   // State in the state machine of the block where the error occurred
      statFBState : DInt := 0;   // State in the state machine of the FB
      statMqttConnectState : DInt := 0;   // State in the state machine of the MQTT Connection
      statMqttCommandState : DInt := 0;   // State in the state machine of the MQTT Commands when MQTT is connected
      statDisablingCompleted : Bool;   // TRUE: Disabling has been completed
      statEmptyDiagnostics : "typeDiagnostics";   // Empty diagnostics information (for initialization purposes only)
      instTsendC : TSEND_C;   // Tsend Instance
      instTrcv : TRCV;   // Trcv Instance
      statSendBuffer : Array[0..#MAX_BUFFER_LEN_SEND] of Byte;   // Send buffer to send Data via TSend
      statRcvBuffer : Array[0..#MAX_BUFFER_LEN_RCV] of Byte;   // Receive buffer to receive Data via Trcv
      statParamQdn : TCON_QDN_SEC;   // Parameter to assign QDN information
      statEmptyParamQdn : TCON_QDN_SEC;   // Empty TCON_QDN_SEC information (for initialization purposes only)
      statParamIp : TCON_IP_V4_SEC;   // Parameter to assign IP information
      statEmptyParamIp : TCON_IP_V4_SEC;   // Empty TCON_IP_V4_SEC information (for initialization purposes only)
      statPublishOld : Bool;   // Old value of 'publish' input for edge detection
      statSubscribeOld : Bool;   // Old value of 'subscribe' input for edge detection
      statUnsubscribeOld : Bool;   // Old value of 'unsubscribe' input for edge detection
      statIsQdn : Bool;   // Static value to set if qdn is used
      statTsendcReq : Bool;   // Static value to set send request
      statTsendcEnable : Bool;   // Static value to set tsend to enabled
      statTsendcLen : UDInt;   // Static value to len of tsend block
      statEnableTimerCommandWatchdog : Bool;   // Static value to start the command timer timeout
      instTimerCommandWatchdog : IEC_TIMER;   // Instance of the Timer for commands
      statEnableMqttKeepAliveTimer : Bool;   // Static value to enable the Mqtt keepalive timer
      statMqttKeepAliveUsed : Bool;   // Static value to show if keepalive is used or deactivated
      statMqttKeepAliveTime : Time;   // Static value to store the keepalive Time interval
      instMqttKeepAliveTimer : IEC_TIMER;   // Instance of the Timer for Mqtt keepalive
      statSendBufferPos : UInt;   // Static value to store the buffer position of the Tsend data area
      statPaketHeaderEncodeDone : Bool;   // Static value to show if a paket header was already encoded
      statSendPaketTotalRemLen : UDInt;   // Static value to store total paket length in bytes
      statEncodedRemPaketLenAsByte : Byte;   // Static value to store remaining length encoded as byte during calculation
      statUsernameLenUtf8Encoded : UInt;   // Static value to store total length of the username in utf8
      statPasswordLenUtf8Encoded : UInt;   // Static value to store total length of the password in utf8
      statWillTopicLenUtf8Encoded : UInt;   // Static value to store total length of the will topic in utf8
      statClientIdLenUtf8Encoded : UInt;   // Static value to store total length of the client id in utf8
      statWillQos : USInt;   // Static value to store the qos information of the will message
      statWillRetain : Bool;   // Static value to store the retain information of the will message
      statWillMessageCnt : UInt;   // Static value to store the amount of valid bytes in will message array
      statClientIdPos : DInt;   // Static value to store client id position during encoding
      statClientIdEncodeState : DInt;   // Static value to store the state during encoding
      statWillMessagePos : DInt;   // Static value to store will message position during encoding
      statWillMessageEncodeState : DInt;   // Static value to store the state during encoding
      statWillTopicPos : DInt;   // Static value to store will topic position during encoding
      statWillTopicEncodeState : DInt;   // Static value to store the state during encoding
      statUserNamePos : DInt;   // Static value to store user name position during encoding
      statUserNameEncodeState : DInt;   // Static value to store the state during encoding
      statPasswordPos : DInt;   // Static value to store password position during encoding
      statPasswordEncodeState : DInt;   // Static value to store the state during encoding
      statPaketId : UInt;   // Static value for the PaketId of each sent paket
      statPublishTopicLenUtf8Encoded : UInt;   // Static value to store total length of the publish topic in utf8
      statPublishQos : USInt;   // Static value to store the qos information of the publish message
      statPublishMessageCnt : UDInt;   // Static value to store the amount of valid bytes in publish message array
      statPublishTopicEncodeState : DInt;   // Static value to store the state during encoding
      statPublishTopicPos : DInt;   // Static value to store publish topic position during encoding
      statPaketIdEncoded : Bool;   // Static value to store if the paket id was encoded
      statPublishEncodeMessageState : DInt;   // Static value to store the state during encoding
      statPublishMessagePos : DInt;   // Static value to store publish message position during encoding
      statSubscribeQos : USInt;   // Static value to store the qos information of the subscribe message
      statSubscribeQosEncoded : Bool;   // Static value to store if the qos was encoded
      statSubscribeTopicPos : DInt;   // Static value to store subscribe topic position during encoding
      statSubscribeTopicEncodeState : DInt;   // Static value to store the state during encoding
      statSubscribeTopicLenUtf8Encoded : UInt;   // Static value to store total length of the subscribe topic in utf8
      statUnsubscribeTopicPos : DInt;   // Static value to store unsubscribe topic position during encoding
      statUnsubscribeTopicEncodeState : DInt;   // Static value to store the state during encoding
      statUnsubscribeTopicLenUtf8Encoded : UInt;   // Static value to store total length of the unsubscribe topic in utf8
      statRcvMsgQoS : UInt;   // Static value to store the qos information of the received message
      statRcvMsgTotalLen : UDInt;   // Static value to store the total len of the received message
      statRcvMsgTopicLen : UInt;   // Static value to store the total len of the received message topic
      statRcvMsgPayloadLen : UDInt;   // Static value to store the total len of the received message payload
      statRcvMsgPaketId : Word;   // Static value to store the paket id of the received message
      statRcvMsgTopicPos : DInt;   // Static value to store received message topic position during decoding
      statRcvMsgPayloadPos : DInt;   // Static value to store received message payload position during decoding
      statRcvMsgDecodeState : DInt;   // State in the state machine of the Rcv decoding
      statRcvMsgInternalStatus : USInt;   // Static value to store the internal status in case of topic or payload overflow
      statSendPubAckMsg : Bool;   // Static value to signal if publish acknowledge message must be sent
   END_VAR
   VAR_TEMP
      tempEnable : Bool;   // Temporary value for input 'enable'
      tempSubscribe : Bool;   // Temporary value for input 'subscribe'
      tempPublish : Bool;   // Temporary value for input 'publish'
      tempUnsubscribe : Bool;   // Temporary value for input 'unsubscribe'
      tempTsendcDone : Bool;   // Temporary value for instance of TsendC
      tempTsendcBusy : Bool;   // Temporary value for instance of TsendC
      tempTsendcError : Bool;   // Temporary value for instance of TsendC
      tempTsendcStatus : Word;   // Temporary value for instance of TsendC
      tempTrcvNdr : Bool;   // Temporary value for instance of Trcv
      tempTrcvBusy : Bool;   // Temporary value for instance of Trcv
      tempTrcvError : Bool;   // Temporary value for instance of Trcv
      tempTrcvStatus : Word;   // Temporary value for instance of Trcv
      tempTrcvRcvdLen : UDInt;   // Temporary value for instance of Trcv
      tempTrcvBufferPos : DInt;   // Temporary value for buffer position in trcv data array
      tempUserFlag : Bool;   // Temporary value to indicate if username is set
      tempPasswordFlag : Bool;   // Temporary value to indicate if passwordis set
      tempWillFlag : Bool;   // Temporary value to indicate if last will is set
      tempWillQoS1 : Bool;   // Temporary value to indicate if lastwill uses qos 1
      tempWillQoS2 : Bool;   // Temporary value to indicate if lastwill uses qos 2
      tempMaxWillMsgLen : DInt;   // Temporary value to store max will msg len
      tempLowerWillMsgArrayBoundary : DInt;   // Temporary value to store will msg data array lower bound from inout
      tempLoopCounter : DInt;   // Temporary value for several For loops
      tempBytesUsedUtf8 : USInt;   // Temporary value to store bytes used by a single character
      tempErrorConvertUtf8 : Bool;   // Temporary value to store if an error occured while converting character to utf8
      tempStatusConvertUtf8 : Word;   // Temporary value to store status code while converting character to utf8
      tempConvertedUtf8 : DWord;   // Temporary value to store the converted character in utf-8 format
      tempWordForSliceAddress : Word;   // Temporary value for several slice accesses
      tempCommandInput : Byte;   // Temporary value to set wether the command was publish subscribe or unsubscribe
      tempRcvMsgTypeCase : Byte;   // Temporary value to store which message type was received
      tempMaxPublishDataArrayLen : DInt;   // Temporary value to store the total length of the publish msg data array at inout
      tempMqttConnAckRcvStatus : USInt;   // Temporary value to store state of connection acknowledgement from broker
      tempMqttPingRspRcv : USInt;   // Temporary value to store PingResponse from broker
      tempMqttPubAckRcv : USInt;   // Temporary value to store Publish acknowledgement of mqtt broker
      tempMqttPubRecRcv : USInt;   // Temporary value to store Publish Received of mqtt broker
      tempMqttPubCompRcv : USInt;   // Temporary value to store Publish Completed of mqtt broker
      tempMqttSubAckRcv : USInt;   // Temporary value to store Subscribe acknowledgement of mqtt broker
      tempMqttUnSubAckRcv : USInt;   // Temporary value to store Unsubscribe acknowledgement of mqtt broker
      tempLowerBoundPublishDataArray : DInt;   // Temporary value to store lower bound of the publish data array
      tempMultiplierToDecode : UDInt;   // Temporary value to store the multiplier while paket decoding algorithm
      tempReceivedTopicStringMaxLen : DInt;   // Temporary value to store the max string len of the received topic
      tempReceivedMsgDataArrayTotalLen : DInt;   // Temporary value to store the total len of the received data msg array at inout
      tempUpperBoundRcvMsgDataArray : DInt;   // Temporary value to store the upper bound of the msg payload array
   END_VAR
   VAR CONSTANT
      FB_STATE_NO_PROCESSING : DInt := 0;   // FB state: No processing
      FB_STATE_VALIDATE_INPUT : DInt := 10;   // FB state: Enabling - Validation of Inputs
      FB_STATE_TCP_CONNECTING : DInt := 20;   // FB state: Processing - TCP Connection establishing
      FB_STATE_OPERATING_MONITOR_TCP : DInt := 30;   // FB state: Processing - TCP Established, MQTT connection in progress
      FB_STATE_TCP_RECONNECTING : DInt := 40;   // FB state: Processing - TCP Connection must be re-established
      FB_STATE_DISABLING : DInt := 90;   // FB state: Disabling
      MQTT_CONNECT_STATE_NO_PROCESSING : DInt := 0;   // MQTT state: No processing
      MQTT_CONNECT_STATE_BUILD_PAKET : DInt := 100;   // MQTT state: Processing - build connect paket
      MQTT_CONNECT_STATE_SEND_PAKET_WAIT_FOR_CONNACK : DInt := 200;   // MQTT state: Processing - send connect paket
      MQTT_CONNECT_STATE_CONNECTED : DInt := 300;   // MQTT state: Processing - Connected to MQTT Broker
      MQTT_CONNECT_STATE_DISCONNECTED : DInt := 400;   // MQTT state: Processing - Disconnected to MQTT Broker
      MQTT_COMMAND_STATE_NO_PROCESSING : DInt := 0;   // MQTT Command state: No processing
      MQTT_COMMAND_STATE_BUILD_PUBLISH : DInt := 1;   // MQTT Command state: Build Publish paket
      MQTT_COMMAND_STATE_SEND_PUBLISH : DInt := 1000;   // MQTT Command state: Send Publish paket
      MQTT_COMMAND_STATE_BUILD_SUBSCRIBE : DInt := 2;   // MQTT Command state: Build Subscribe paket
      MQTT_COMMAND_STATE_SEND_SUBSCRIBE : DInt := 2000;   // MQTT Command state: Send Subscribe paket
      MQTT_COMMAND_STATE_BUILD_UNSUBSCRIBE : DInt := 4;   // MQTT Command state: Build Unsubscribe paket
      MQTT_COMMAND_STATE_SEND_UNSUBSCRIBE : DInt := 3000;   // MQTT Command state: Send Unsubscribe paket
      MQTT_COMMAND_STATE_SEND_PING : DInt := 8000;   // MQTT Command state: Send Ping paket
      MQTT_COMMAND_STATE_PING_RESP : DInt := 9000;   // MQTT Command state: Receive Ping paket
      STATUS_JOB_EXECUTED : Word := 16#0000;   // The last job was successfully executed
      STATUS_NO_CALL : Word := 16#7000;   // No job being currently processed
      STATUS_FIRST_CALL : Word := 16#7001;   // First call after incoming new job (rising edge 'enable')
      STATUS_SUBSEQUENT_CALL : Word := 16#7002;   // Subsequent call during active processing without further details
      STATUS_MQTT_CONNECTING : Word := 16#7003;   // Currently connecting to MQTT Broker
      STATUS_MQTT_CONNECTED : Word := 16#7004;   // Connected to MQTT Broker
      STATUS_MQTT_PING : Word := 16#7005;   // Processing Ping to Broker
      STATUS_MQTT_PUBLISH : Word := 16#7006;   // Processing Publish to Broker
      STATUS_MQTT_SUBSCRIBE : Word := 16#7008;   // Processing Subscribe to Broker
      STATUS_MQTT_UNSUBSCRIBE : Word := 16#7010;   // Processing Unsubscribe to Broker
      ERR_UNDEFINED_STATE : Word := 16#8600;   // Error due to an undefined state in state machine
      ERR_TCP_RECONNECTING : Word := 16#9000;   // Error, lost connection to mqtt broker, reconnect ongoing
      ERR_CLIENT_ID_NULL : Word := 16#8200;   // Error due to an incorrect client id at input
      ERR_CNT_EXCEEDS_ARRAY_DIMENSION : Word := 16#8210;   // Error due to an incorrect assignment of publish msg len or will msg len
      ERR_KEEPALIVE_INVALID : Word := 16#8220;   // Error due to an incorrect assignment of keepalive input
      ERR_QOS_INVALID : Word := 16#8230;   // Error due to an incorrect assignment of qos input
      ERR_TCON_FAILED : Word := 16#8601;   // Error while trying to connect to mqtt broker with tcon
      ERR_TCON_TIMEOUT : Word := 16#8620;   // Error due to time out while trying to connect to broker
      ERR_MQTT_REM_LEN_INVALID : Word := 16#8700;   // Error due to receiving an invalid mqtt paket
      ERR_MQTT_MALFORMED_QOS_RECEIVED : Word := 16#8710;   // Error due to receiving an invalid mqtt paket
      ERR_MQTT_CONNACK_INVALID_SESSION_FLAG : Word := 16#8720;   // Error due to receiving an invalid mqtt paket
      ERR_MQTT_CONNACK_RETURN_CODE_INVALID : Word := 16#8730;   // Error due to receiving an invalid mqtt paket - see subfunction status for more information
      ERR_MQTT_PAKET_ID_INVALID : Word := 16#8740;   // Error due to receiving an invalid mqtt paket id
      ERR_MQTT_SUBACK_FAILURE : Word := 16#8750;   // Error because of failing to create a subscription
      ERR_MQTT_COMMAND_MULTIPLE_INPUT : Word := 16#8001;   // Error - wrong operation - simultaneous input
      ERR_MQTT_COMMAND_PUBLISH_TOPIC_INVALID : Word := 16#8300;   // Error - publish topic empty or invalid
      ERR_MQTT_COMMAND_SUBSCRIBE_TOPIC_INVALID : Word := 16#8310;   // Error - subscribe topic empty or invalid
      ERR_MQTT_COMMAND_UNSUBSCRIBE_TOPIC_INVALID : Word := 16#8320;   // Error - unsubscribe topic empty or invalid
      ERR_MQTT_COMMAND_SEND_TIMEOUT : Word := 16#8650;   // Error - timeout while trying to sending data
      ERR_MQTT_CONNECT_TIMEOUT : Word := 16#8670;   // Error - timout while trying to connect via mqtt to broker
      MAX_BUFFER_LEN_RCV : UInt := 1459;   // Max. Buffer Len for TRCV
      MAX_BUFFER_LEN_SEND : UInt := 8191;   // Max. Buffer Len for TSEND on S7-1200/S7-1500
      EMPTY_BYTE : Byte := 16#00;   // Empty byte for initalisation
      NO_COMMAND : Byte := 16#00;   // No Command for Executing Publish, Subscribe, Unsubscribe
      EMPTY_STRING : String;   // Empty string for initalisation
      EMPTY_WSTRING : WString;   // Empty wstring for initalisation
      LEN_NULL : Int := 0;   // Integer 0 to compare length to zero
      INIT_UDINT_1 : UDInt := 1;   // Udint with value 1 for initalisation
      ARRAY_LEN_OFFSET_PLUS_1 : DInt := 1;   // Offset for array boundaries
      FIRST_CHARACTER : DInt := 1;   // First character in a character string
      ONE_DIMENSION : UDInt := 1;   // one dimensional array
      FIRST_ENCODING : DInt := 1;   // First encoding state while encoding messages
      SUBSEQUENT_ENCODING : DInt := 2;   // Followig encoding state while encoding messages if it takes multiple cycles
      ENCODE_DONE : DInt := 3;   // Last encoding state while encoding messages
      NOT_USED_NO_ENCODING : DInt := 5;   // No encoding state while encoding messages
      MSG_DECODE_STATE_NO_PROCESSING : DInt := 0;   // No message processing
      MSG_DECODE_STATE_TOPIC : DInt := 1;   // Message decoding state for topic
      MSG_DECODE_STATE_PAKET_ID_MSB : DInt := 2;   // Message decoding state for paket id msb
      MSG_DECODE_STATE_PAKET_ID_LSB : DInt := 3;   // Message decoding state for paket id lsb
      MSG_DECODE_STATE_PAYLOAD : DInt := 4;   // Message decoding state for paket payload
      MSG_DECODE_STATUS_NO_NEW_MSG : USInt := 0;   // Message decoding status if no new message was received
      MSG_DECODE_STATUS_NEW_MSG_OK : USInt := 1;   // Message decoding status if anew message was received
      MSG_DECODE_STATUS_TOPIC_TOO_LONG : USInt := 2;   // Message decoding status if new message was received bute topic does not fit it inout topic (too shoirt)
      MSG_DECODE_STATUS_PAYLOAD_TOO_LONG : USInt := 2;   // Message decoding status if new message was received bute payload does not fit it inout payload(too shoirt)
      MQTT_QOS_0 : UInt := 0;   // Saving mqtt qos 0
      MQTT_QOS_1 : UInt := 1;   // Saving mqtt qos 1
      MQTT_QOS_2 : UInt := 2;   // Saving mqtt qos 2
      REMAINING_LEN_3 : Byte := 16#03;   // Remaining len in bytes is 3
      REMAINING_LEN_2 : Byte := 16#02;   // Remaining len in bytes is 2
      REMAINIG_LEN_0 : Byte := 16#00;   // Remaining len in bytes is 0
      SUBSCRIBE_FAILURE : Byte := 16#80;   // Subscription failed flag.
      MQTT_NO_SESSION_PRESENT : Byte := 16#00;   // No session present indication
      KEEPALIVE_DISABLED : Time := t#0s;   // Mqtt keepalive set to 0s
      TSENDC_JOB_DONE : Word := 16#0000;   // Status of tsendc if job was successful
      TSENDC_COM_CLOSED : Word := 16#0003;   // Status of tsendc if connection closed
      TSENDC_EST_OK : Word := 16#7004;   // Status of tsendc if connection ok
      TSENDC_DISCONNECTED : Word := 16#7000;   // Status of tsendc if disconnected from broker
      UINT_CONST_1000 : UInt := 1000;   // Calculation to seconds
      TWO_SECONDS : UInt := 2000;   // Calculation by 2 seconds
      THREE_SECONDS : UInt := 3;   // Upper limit is 3 seconds
      UTF_1_BYTE_USED : USInt := 1;   // If utf uses 1 byte
      UTF_2_BYTE_USED : USInt := 2;   // If utf uses 2 byte
      UTF_3_BYTE_USED : USInt := 3;   // If utf uses 3 byte
      ONE_BYTE_LEN_INFO : UInt := 1;   // Adds one byte len info
      TWO_BYTE_LEN_INFO : UInt := 2;   // Adds two byte len info
      CONNECT_HEADER_10BYTE_LEN : UInt := 10;   // Connect header has always 10 byte minimum
      NO_RESPONSE : USInt := 0;   // If no response received from broker
      RESPONSE_GOOD : USInt := 1;   // If good response received from broker
      RESPONSE_PAKET_ID_INVALID : USInt := 2;   // If response received from broker but paket id invalid
      RESPONSE_SUBSCRIBE_FAILED : USInt := 3;   // If response received from broker but subscribption invalid
      MQTT_MSG_TYPE_CONNECT : Byte := 16#10;   // CONNECT MQTT Control Packet (see MQTT standard for more info)
      MQTT_MSG_TYPE_CONNACK : Byte := 16#20;   // CONNACK MQTT Control Packet (see MQTT standard for more info)
      MQTT_MSG_TYPE_DISCONNECT : Byte := 16#E0;   // DISCONNECT MQTT Control Packet (see MQTT standard for more info)
      MQTT_MSG_TYPE_PUBLISH : Byte := 16#30;   // PUBLISH MQTT Control Packet for QoS = 0 (see MQTT standard for more info)
      MQTT_MSG_TYPE_PUBACK : Byte := 16#40;   // PUBACK MQTT Control Packet (see MQTT standard for more info)
      MQTT_MSG_TYPE_PUBREC : Byte := 16#50;   // PUBREC MQTT Control Packet (see MQTT standard for more info)
      MQTT_MSG_TYPE_PUBREL : Byte := 16#62;   // PUBREL MQTT Control Packet (see MQTT standard for more info)
      MQTT_MSG_TYPE_PUBCOMP : Byte := 16#70;   // PUBCOM MQTT Control Packet (see MQTT standard for more info)
      MQTT_MSG_TYPE_SUBSCRIBE : Byte := 16#82;   // SUBSCRIBE MQTT Control Packet (see MQTT standard for more info)
      MQTT_MSG_TYPE_UNSUBSCRIBE : Byte := 16#A2;   // UNSUBSCRIBE MQTT Control Packet (see MQTT standard for more info)
      MQTT_MSG_TYPE_SUBACK : Byte := 16#90;   // SUBACK MQTT Control Packet (see MQTT standard for more info)
      MQTT_MSG_TYPE_UNSUBACK : Byte := 16#B0;   // UNSUBACK MQTT Control Packet (see MQTT standard for more info)
      MQTT_MSG_TYPE_PING : Byte := 16#C0;   // PING MQTT Control Packet (see MQTT standard for more info)
      MQTT_MSG_TYPE_PINGRESP : Byte := 16#D0;   // PINGRESP MQTT Control Packet (see MQTT standard for more info)
      MQTT_MSG_TYPE_RCV_PUB_MESSAGE : Byte := 16#30;   // PUBLISH MQTT Control Packet for QoS = 0 (see MQTT standard for more info)
      MQTT_MSG_TYPE_RCV_PUB_MESSAGE_QoS0 : Byte := 16#30;   // PUBLISH MQTT Control Packet for QoS = 0 (see MQTT standard for more info)
      MQTT_MSG_TYPE_RCV_PUB_MESSAGE_QoS1 : Byte := 16#32;   // PUBLISH MQTT Control Packet for QoS = 1 (see MQTT standard for more info)
      MQTT_MSG_TYPE_RCV_PUB_MESSAGE_QoS2 : Byte := 16#34;   // PUBLISH MQTT Control Packet for QoS = 2 (see MQTT standard for more info)
      MQTT_MSG_TYPE_RCV_PUB_MESSAGE_BAD : Byte := 16#36;   // PUBLISH MQTT Control Packet for QoS =1 and QoS=2 at the same time (see MQTT standard for more info)
      MQTT_MSG_DECODING : Byte := 16#FF;   // STATE to show that currently a message is being decoded
      MQTT_CONNACK_ACCEPTED : Byte := 16#00;   // Connect acknowledge flag in case no session present flag was not set
      BIT_MASK_HIGHBITS : Byte := 16#F0;   // MQTT Message Types only use High bits, so we only use High bits and ignore low bits
      BIT_MASK_QOS : Byte := 16#F6;   // A Bit Mask to only validate recieved Byte against QOS Value
      DEFAULT_VALUE_ZERO : Int := 0;   // DEFAULT Value for Variables that a ZERO Based
      SEND_LEN_MULTIPLIER_UDINT_128 : UDInt := 128;   // Default mulitplier to calculate package length
      MAX_ALLOWED_PAKET_SIZE : UDInt := 2097152;   // The highest amount of payload to be sent by mqtt paket
      DEFAULT_MULTIPLIER_BYTE_127 : Byte := 16#7F;   // Default mulitplier to calculate package length
      CONN_PROTOCOL_NAME_0 : Byte := 16#00;   // Protocol version for mqtt
      CONN_PROTOCOL_NAME_4 : Byte := 16#04;   // Protocol version for mqtt
      CONN_PROTOCOL_MQTT_VERSION_3_1_1 : Byte := 16#04;   // Protocol version for mqtt
   END_VAR
BEGIN
   REGION BLOCK INFO HEADER
     //===============================================================================
     // SIEMENS / (c)Copyright 2020
     //-------------------------------------------------------------------------------
     // Title:        LMQTT_Client
     // Function:     This FB implements an MQTT client. A user can publish data and
     //               subscribe to topics to receive data.
     // Library:      LMQTT
     // Author:       Siemens Industry Online Support
     // Tested with:  CPU 1516-3 PN/DP FW 2.8
     // Engineering:  TIA Portal V16
     // Restrictions: --
     // Requirements: S7-1200 with firmware V4.4 or higher
     //               S7-1500 with firmware V2.0 or higher
     //-------------------------------------------------------------------------------
     // Change log table:
     // Version  | Date       | Expert in charge       | Changes applied
     //----------|------------|------------------------|------------------------------
     // 01.00.00 | 2017-06-06 | Online Support         | First released version
     // 02.00.00 | 2018-06-04 | Online Support         | Added DNS support and Subscribe to topics
     // 02.01.00 | 2019-11-10 | Online Support         | Minor connection improvements. Updated some comments
     // 02.02.01 | 2019-12-03 | Online Support         | Update to V16 and fusion with S7-1200 Lib
     // 02.02.02 | 2020-03-16 | Online Support         | Improved issue with validateSubjectAlternateNameOfServer
     //          |            |                        | not setting correct bit
     // 03.00.00 | 2020-11-04 | Online Support         | New block interface with major improvements
     // 03.00.03 | 2021-05-07 | Online Support         | Minor bug fixes
     //===============================================================================
   END_REGION

   #tempEnable := #enable; // Work with temporary value / create process image
   #tempPublish := #publish;  // Work with temporary value / create process image - only checked when MQTT is connected
   #tempSubscribe := #subscribe;  // Work with temporary value / create process image - only checked when MQTT is connected
   #tempUnsubscribe := #unsubscribe;  // Work with temporary value / create process image - only checked when MQTT is connected


   REGION OUC_BLOCK_CALLS
     //Only call if FB is processing
     IF #statStatus <> #STATUS_NO_CALL THEN
       // Connect and send
       IF #statIsQdn = TRUE THEN // Call if host is a domain name
         #instTsendC(REQ     := #statTsendcReq,
                     CONT    := #statTsendcEnable,
                     LEN     := #statTsendcLen,
                     DONE    => #tempTsendcDone,
                     BUSY    => #tempTsendcBusy,
                     ERROR   => #tempTsendcError,
                     STATUS  => #tempTsendcStatus,
                     CONNECT := #statParamQdn,
                     DATA    := #statSendBuffer);

       ELSE
         #instTsendC(REQ     := #statTsendcReq,
                     CONT    := #statTsendcEnable,
                     LEN     := #statTsendcLen,
                     DONE    => #tempTsendcDone,
                     BUSY    => #tempTsendcBusy,
                     ERROR   => #tempTsendcError,
                     STATUS  => #tempTsendcStatus,
                     CONNECT := #statParamIp,
                     DATA    := #statSendBuffer);
       END_IF;

       // Receive only when TCP operating
       #instTrcv(EN_R     := (#statFBState = #FB_STATE_OPERATING_MONITOR_TCP),
                 ID       := #statParamQdn.ConnPara.ID,
                 ADHOC    := true,
                 NDR      => #tempTrcvNdr,
                 BUSY     => #tempTrcvBusy,
                 ERROR    => #tempTrcvError,
                 STATUS   => #tempTrcvStatus,
                 RCVD_LEN => #tempTrcvRcvdLen,
                 DATA     := #statRcvBuffer);

       //Monitor Time out
       #instTimerCommandWatchdog.TON(IN := #statEnableTimerCommandWatchdog,
                                 PT := #timeOut);
       //Mqtt Keepalive Timer
       #instMqttKeepAliveTimer.TON(IN := #statEnableMqttKeepAliveTimer,
                               PT := #statMqttKeepAliveTime);


     END_IF;
   END_REGION


   REGION ENABLING/DISABLING_FUNCTION_BLOCK
     IF (#tempEnable = TRUE) AND (#statStatus = #STATUS_NO_CALL) THEN // Enable FB
       // First call; initialize FB
       #statValid := TRUE;
       #statBusy := TRUE;
       #statError := FALSE;
       #statDone := FALSE;
       #statErrorUserCleared := FALSE;
       #statErrorAutoCleared := FALSE;
       #statStatus := #STATUS_FIRST_CALL;
       #statSubfunctionStatus := #STATUS_JOB_EXECUTED;
       #statFBErrorState := 0;
       #diagnostics := #statEmptyDiagnostics;
       #statDisablingCompleted := FALSE;
       // State machine - start functionality
       #statFBState := #FB_STATE_VALIDATE_INPUT;

       // Initialize functionality: reset of variables, diagnostics, etc.
       #statPublishOld := FALSE;
       #statSubscribeOld := FALSE;
       #statUnsubscribeOld := FALSE;
       #statIsQdn := FALSE;
       #statTsendcReq := FALSE;
       #statTsendcEnable := FALSE;
       #statPaketHeaderEncodeDone := FALSE;
       #statTsendcLen := 0;
       #statParamQdn := #statEmptyParamQdn;
       #statParamIp := #statEmptyParamIp;
       #statEnableTimerCommandWatchdog := FALSE;
       #statEnableMqttKeepAliveTimer := FALSE;
       #statSendBufferPos := 0;
       #statPaketId := 0;
       #statPublishQos := 0;
       #statWillQos := 0;
       #statWillRetain := FALSE;
       #statWillMessageCnt := 0;
       #statMqttKeepAliveTime := #KEEPALIVE_DISABLED;
       #statMqttKeepAliveUsed := FALSE;
       #statSendBufferPos := 0;
       #statPaketHeaderEncodeDone := FALSE;
       #statSendPaketTotalRemLen := 0;
       #statEncodedRemPaketLenAsByte := #EMPTY_BYTE;
       #statUsernameLenUtf8Encoded := 0;
       #statPasswordLenUtf8Encoded := 0;
       #statWillTopicLenUtf8Encoded := 0;
       #statClientIdLenUtf8Encoded := 0;
       #statWillQos := 0;
       #statWillRetain := FALSE;
       #statWillMessageCnt := 0;
       #statClientIdPos := 0;
       #statClientIdEncodeState := 0;
       #statWillMessagePos := 0;
       #statWillMessageEncodeState := #FIRST_ENCODING;
       #statWillTopicPos := 0;
       #statWillTopicEncodeState := #FIRST_ENCODING;
       #statUserNamePos := 0;
       #statUserNameEncodeState := #FIRST_ENCODING;
       #statPasswordPos := 0;
       #statPasswordEncodeState := #FIRST_ENCODING;
       #statPaketId := 0;
       #statPublishTopicLenUtf8Encoded := 0;
       #statPublishQos := 0;
       #statPublishMessageCnt := 0;
       #statPublishTopicEncodeState := #FIRST_ENCODING;
       #statPublishTopicPos := 0;
       #statPaketIdEncoded := FALSE;
       #statPublishEncodeMessageState := #FIRST_ENCODING;
       #statPublishMessagePos := 0;
       #statSubscribeQos := 0;
       #statSubscribeQosEncoded := FALSE;
       #statSubscribeTopicPos := 0;
       #statSubscribeTopicEncodeState := #FIRST_ENCODING;
       #statSubscribeTopicLenUtf8Encoded := 0;
       #statUnsubscribeTopicPos := 0;
       #statUnsubscribeTopicEncodeState := #FIRST_ENCODING;
       #statUnsubscribeTopicLenUtf8Encoded := 0;
       #statRcvMsgQoS := 0;
       #statRcvMsgTotalLen := 0;
       #statRcvMsgTopicLen := 0;
       #statRcvMsgPayloadLen := 0;
       #statRcvMsgPaketId := 0;
       #statRcvMsgTopicPos := 0;
       #statRcvMsgPayloadPos := 0;
       #statRcvMsgDecodeState := #MSG_DECODE_STATE_NO_PROCESSING;
       #statRcvMsgInternalStatus := 0;
       #statRcvMsgStatus := 0;
       #statRcvMsgDataLen := 0;
       #statSendPubAckMsg := FALSE;

       // Initialize functionality: call subsidiary FBs with FALSE
       FILL_BLK(IN    := #EMPTY_BYTE,
                COUNT := #MAX_BUFFER_LEN_SEND,
                OUT   => #statSendBuffer[0]);
       FILL_BLK(IN    := #EMPTY_BYTE,
                COUNT := #MAX_BUFFER_LEN_RCV,
                OUT   => #statRcvBuffer[0]);
       RESET_TIMER(#instTimerCommandWatchdog);
       RESET_TIMER(#instMqttKeepAliveTimer);

       // INIT SUB STATE MACHINES
       #statMqttConnectState := #MQTT_CONNECT_STATE_NO_PROCESSING;
       #statMqttCommandState := #MQTT_COMMAND_STATE_NO_PROCESSING;
       #statRcvMsgDecodeState := #MSG_DECODE_STATE_NO_PROCESSING;

     ELSIF (#tempEnable = FALSE) AND (#statEnableOld = TRUE) THEN // Disable FB 
       #statFBState := #FB_STATE_DISABLING;
     ELSIF (#statStatus = #STATUS_FIRST_CALL) THEN // Set status identifier of subsequent call
       #statStatus := #STATUS_SUBSEQUENT_CALL;
     END_IF;

     // Edge detection 'enable' input
     #statEnableOld := #tempEnable;
   END_REGION ENABLING/DISABLING

   IF (#statStatus = #STATUS_NO_CALL) THEN // Nothing to do -> End here to reduce "system load"
     RETURN;
   END_IF;

   REGION STATE_MACHINE_FUNCTION_BLOCK_TCP
     CASE #statFBState OF // State machine of FB
       #FB_STATE_NO_PROCESSING: // No processing active (Note: this state must always be present and left empty)
         ;

       #FB_STATE_VALIDATE_INPUT: // Enabling active
         REGION FB_VALIDATE_INPUT
           #statParamIp.ConnPara.ID := #connParam.connId;
           #statParamQdn.ConnPara.ID := #connParam.connId;

           #statParamIp.ConnPara.InterfaceId := #connParam.hwId;
           #statParamQdn.ConnPara.InterfaceId := #connParam.hwId;

           #statParamIp.ConnPara.ActiveEstablished := TRUE;
           #statParamQdn.ConnPara.ActiveEstablished := TRUE;

           #statParamQdn.ConnPara.RemotePort := #connParam.brokerAddress."port";
           #statParamIp.ConnPara.RemotePort := #connParam.brokerAddress."port";

           IF #connParam.tls.enableTls THEN
             #statParamQdn.ActivateSecureConn := TRUE;
             #statParamIp.ActivateSecureConn := TRUE;

             #statParamQdn.TLSServerCertRef := #connParam.tls.brokerCert;
             #statParamIp.TLSServerCertRef := #connParam.tls.brokerCert;

             #statParamQdn.TLSClientCertRef := #connParam.tls.clientCert;
             #statParamIp.TLSClientCertRef := #connParam.tls.clientCert;

             #statParamQdn.ExtTLSCapabilities.%X0 := #connParam.tls.validateServerIdentity;
             #statParamIp.ExtTLSCapabilities.%X0 := #connParam.tls.validateServerIdentity;
           END_IF;

           IF #connParam.brokerAddress.qdnAddress <> #EMPTY_STRING THEN
             #statIsQdn := TRUE;
             #statParamQdn.ConnPara.RemoteQDN := #connParam.brokerAddress.qdnAddress;
           ELSE
             #statIsQdn := FALSE;
             #statParamIp.ConnPara.RemoteAddress.ADDR[1] := #connParam.brokerAddress.ipAddress.ADDR[1];
             #statParamIp.ConnPara.RemoteAddress.ADDR[2] := #connParam.brokerAddress.ipAddress.ADDR[2];
             #statParamIp.ConnPara.RemoteAddress.ADDR[3] := #connParam.brokerAddress.ipAddress.ADDR[3];
             #statParamIp.ConnPara.RemoteAddress.ADDR[4] := #connParam.brokerAddress.ipAddress.ADDR[4];
           END_IF;

           //Check Input variables:
           #tempMaxWillMsgLen := ABS(UPPER_BOUND(ARR := #willMsgPayload, DIM := #ONE_DIMENSION) - LOWER_BOUND(ARR := #willMsgPayload, DIM := #ONE_DIMENSION)) + #ARRAY_LEN_OFFSET_PLUS_1;


           //Check Client ID len Must be > 0 
           IF LEN(#clientIdentifier) <= #LEN_NULL THEN
             #statStatus := #ERR_CLIENT_ID_NULL; // Set correct status that identifies error clearly
             #statSubfunctionStatus := #ERR_CLIENT_ID_NULL; // Status or return value of called FBs, FCs and system blocks
             #statFBErrorState := #statFBState; // Set error state number for diagnostic 
             #statErrorUserCleared := TRUE;
             //verify Will next
           ELSIF #tempMaxWillMsgLen < #willMsgLen THEN
             #statStatus := #ERR_CNT_EXCEEDS_ARRAY_DIMENSION; // Set correct status that identifies error clearly
             #statSubfunctionStatus := #ERR_CNT_EXCEEDS_ARRAY_DIMENSION; // Status or return value of called FBs, FCs and system blocks
             #statFBErrorState := #statFBState; // Set error state number for diagnostic 
             #statErrorUserCleared := TRUE;
             ///CHECK WILL QOS
           ELSIF #qos > #MQTT_QOS_2 THEN
             #statStatus := #ERR_QOS_INVALID; // Set correct status that identifies error clearly
             #statSubfunctionStatus := #ERR_QOS_INVALID; // Status or return value of called FBs, FCs and system blocks
             #statFBErrorState := #statFBState; // Set error state number for diagnostic 
             #statErrorUserCleared := TRUE;
           ELSIF (#connParam.keepAlive < #THREE_SECONDS) // IF Set to 1 or 2 seconds..
             AND (#connParam.keepAlive > 0)
           THEN
             #statStatus := #ERR_KEEPALIVE_INVALID; // Set correct status that identifies error clearly
             #statSubfunctionStatus := #ERR_KEEPALIVE_INVALID; // Status or return value of called FBs, FCs and system blocks
             #statFBErrorState := #statFBState; // Set error state number for diagnostic 
             #statErrorUserCleared := TRUE;
           ELSE
             //Set Params for connection
             //Set Client Id
             #statWillQos := #qos;
             //set Retain
             #statWillRetain := #retain;
             // Will message cnt
             #statWillMessageCnt := #willMsgLen;
             //Keepalive
             IF #connParam.keepAlive = 0 THEN
               #statMqttKeepAliveUsed := FALSE;
             ELSE
               #statMqttKeepAliveUsed := TRUE;
               //KeepAliveTImer is set to ((Keep Alive converted to seconds) - 2s)
               #statMqttKeepAliveTime := UINT_TO_TIME((#connParam.keepAlive * #UINT_CONST_1000 - #TWO_SECONDS));
             END_IF;
             //rdy to enable TCON
             #statTsendcEnable := TRUE;
             #statEnableTimerCommandWatchdog := TRUE;
             #statFBState := #FB_STATE_TCP_CONNECTING;
           END_IF;
         END_REGION FB_VALIDATE_INPUT

       #FB_STATE_TCP_CONNECTING: //Wait for TCP to be established
         REGION FB_TCP_CONNECTING
           //Check process:
           IF #tempTsendcError = TRUE THEN //when error:
             #statTsendcEnable := FALSE; //disable TsendC
             #statEnableTimerCommandWatchdog := FALSE;
             #statStatus := #ERR_TCON_FAILED; // Set correct status that identifies error clearly
             #statSubfunctionStatus := #tempTsendcStatus; // Status or return value of called FBs, FCs and system blocks
             #statFBErrorState := #statFBState; // Set error state number for diagnostic 
             #statErrorUserCleared := TRUE;
           ELSIF #tempTsendcStatus = #TSENDC_EST_OK THEN //when successfull:
             //     Communication connection established.
             #statEnableTimerCommandWatchdog := FALSE;
             //Monitor Connection
             #statFBState := #FB_STATE_OPERATING_MONITOR_TCP;
             // Begin MQTT Connection
             #statMqttConnectState := #MQTT_CONNECT_STATE_BUILD_PAKET;
             //set status
             #statStatus := #STATUS_MQTT_CONNECTING;
           ELSIF #instTimerCommandWatchdog.Q THEN
             #statTsendcEnable := FALSE; //disable TsendC
             #statEnableTimerCommandWatchdog := FALSE;
             #statStatus := #ERR_TCON_TIMEOUT; // Set correct status that identifies error clearly
             #statSubfunctionStatus := #ERR_TCON_TIMEOUT; // Status or return value of called FBs, FCs and system blocks
             #statFBErrorState := #statFBState; // Set error state number for diagnostic 
             #statErrorUserCleared := TRUE;
           END_IF;
         END_REGION FB_TCP_CONNECTING
       #FB_STATE_OPERATING_MONITOR_TCP: // Processing active
         REGION FB_OPERATING_MONITOR_TCP
           //Reset Status on Msg Output - will be set when a new message is completly processed and ready at outputs.
           #statRcvMsgStatus := #MSG_DECODE_STATUS_NO_NEW_MSG;
           //Reset TsendC Req from last  cycle Request:
           #statTsendcReq := FALSE;
           //Monitor Connection - if disconnect occured:
           IF ((#tempTsendcStatus > #TSENDC_COM_CLOSED AND #tempTsendcStatus < #TSENDC_EST_OK) //Status connection interupt
             OR #tempTsendcError = TRUE) // Or error
             AND #tempTrcvNdr = FALSE // And no new data (to see if broker send information why connection was interrupted)
           THEN
             REGION CONNECTION_INTERRUPTED
               //Status reconnecting
               //SET MQTT to no operation
               #statMqttConnectState := #MQTT_CONNECT_STATE_NO_PROCESSING;
               #statMqttCommandState := #MQTT_COMMAND_STATE_NO_PROCESSING;
               #statRcvMsgDecodeState := #MSG_DECODE_STATE_NO_PROCESSING;
               //Reset Pub ack
               #statSendPubAckMsg := FALSE;
               //reset Done bit if still set, regardless of input:
               #statDone := FALSE;
               //reset Watchdog
               #statEnableTimerCommandWatchdog := FALSE;
               // reset headerEncode
               #statPaketHeaderEncodeDone := FALSE;
               //set error  information
               #statStatus := #ERR_TCP_RECONNECTING; // Set correct status that identifies error clearly
               #statSubfunctionStatus := #tempTsendcStatus;// Status or return value of called FBs, FCs and system blocks
               #statFBErrorState := #statFBState; // Set error state number for diagnostic 
               #statErrorAutoCleared := TRUE;
               //Wait for reconect - next state
               #statFBState := #FB_STATE_TCP_RECONNECTING;
             END_REGION REGION CONNECTION_INTERRUPTED
           ELSE
             //Connection is OK
             //Sending and receiving works 
             //Check Trcv Buffer for new Data
             IF #tempTrcvNdr THEN
               REGION TRCV_NEW_DATA
                 //Evaluate the TrcvBuffer, reset buffer pos to start
                 #tempTrcvBufferPos := 0;
                 // Parse the whole RCV Buffer
                 WHILE #tempTrcvBufferPos < (UDINT_TO_DINT(#tempTrcvRcvdLen)) DO
                   // Parse the whole RCV Buffer, check wether header or decoding
                   IF #statRcvMsgDecodeState = #MSG_DECODE_STATE_NO_PROCESSING THEN
                     //If no decoding is in progress, look for new message header
                     #tempRcvMsgTypeCase := #statRcvBuffer[#tempTrcvBufferPos] AND #BIT_MASK_HIGHBITS;
                   ELSE
                     //decode is in progress, go directly to decoding
                     #tempRcvMsgTypeCase := #MQTT_MSG_DECODING;
                   END_IF;

